(* PLC project Scenario24, Beckhoff Automation GmbH TwinCAT PLC Control 3.5.8.40 *)
(* stored: creationDateTime 2018-05-29T16:20:14.9693905, modificationDateTime 2018-05-29T16:20:14.9929599 *)

TYPE RFID_ByteArray :
STRUCT
	RFID_Data : ARRAY[0..127] OF BYTE;
END_STRUCT
END_TYPE

PROGRAM MAIN
VAR		
	xPPU : xPPU;

//Stack
	//Waiting for Signals
	Check_Stack_WPPickedUp :BOOL;	
	//Giving Signals
	Stack_WPProvided : BOOL;
	Stack_WPType_Black : BOOL;
	Stack_WPType_White : BOOL;
	Stack_WPType_Metallic : BOOL;
	Stack_WPWeight_Light : BOOL;
	Stack_WPWeight_Medium : BOOL;
	Stack_WPWeight_Heavy : BOOL;
//Crane
	//Waiting for Signals
	Check_Stack_WPProvided : BOOL;
	Check_Stack_WPType_Black : BOOL;
	Check_Stack_WPType_White : BOOL;
	Check_Stack_WPType_Metallic : BOOL;
	Check_LargeSortingConveyor_IsSorting : BOOL;
	Check_LargeSortingConveyor_AutomaticExecuteCompleted : BOOL;	
	Check_Stamp_IsStamping : BOOL;
	Check_Stamp_WPAvailable : BOOL;
	Check_Stamp_AutomaticExecuteCompleted : BOOL;
	Check_RefillConveyor_IsSending : BOOL;
	//Giving Signals
	Crane_WPType_Black : BOOL;
	Crane_WPType_White : BOOL;
	Crane_WPType_Metallic : BOOL;
	Crane_WPWeight_Light : BOOL;
	Crane_WPWeight_Medium : BOOL;
	Crane_WPWeight_Heavy : BOOL;
	Crane_Conveyor_AllowedToOperate : BOOL;
	Crane_Stamp_AllowedToOperate : BOOL;
	Crane_WPPickedUp : BOOL;
//Stamp	
	//Waiting for Signals
	Check_Stamp_AllowedToOperate : BOOL;
	Check_Stamp_WPWeight_Light : BOOL;
	Check_Stamp_WPWeight_Medium : BOOL;
    Check_Stamp_WPWeight_Heavy : BOOL;
	//Giving Signals
	Stamp_WPType_Black : BOOL;
	Stamp_WPType_White : BOOL;
	Stamp_WPType_Metallic : BOOL;
	Stamp_WPWeight_Light : BOOL;
	Stamp_WPWeight_Medium : BOOL;
	Stamp_WPWeight_Heavy : BOOL;
	Stamp_IsStamping : BOOL;
	Stamp_WPAvailable : BOOL;
	Stamp_AutomaticExecuteCompleted	: BOOL;
//LargeSortingConveyor
	//Waiting for Signals
	Check_LargeSortingConveyor_AllowedToOperate : BOOL;
	Check_LargeSortingConveyor_FollowConveyorInitCompleted : BOOL;	
	Check_LargeSortingConveyor_FollowConveyorAutoamticExecuteCompleted : BOOL;	
	//Giving Signals	
	LargeSortingConveyor_InitCompleted : BOOL;
	LargeSortingConveyor_NumberOfWPsAtConveyor : USINT;
	LargeSortingConveyor_FollowConveyor_AllowedToInit : BOOL;
	LargeSortingConveyor_FollowConveyor_AllowedToOperate: BOOL;
	LargeSortingConveyor_IsSorting : BOOL;
	LargeSortingConveyor_AutomaticExecuteCompleted : BOOL;	
//PicALphaConveyor
	//Waiting for Signals
	Check_PicAlphaConveyor_AllowedToInit : BOOL;
	Check_PicAlphaConveyor_AllowedToReceive : BOOL;
	Check_PicAlphaConveyor_AllowedToSend : BOOL;
	Check_PicAlphaConveyor_FollowConveyor_InitCompleted : BOOL;
	Check_PicAlphaConveyor_PicAlpha_AutomaticExecuteCompleted : BOOL;
	Check_PicAlphaConveyor_FollowConveyor_AutomaticExecuteCompleted : BOOL;
	//Giving Signals
	PicAlphaConveyor_InitCompleted : BOOL;
	PicAlphaConveyor_FollowConveyor_AllowedToInit : BOOL;
	PicAlphaConveyor_PicAlpha_AllowedToOperate : BOOL;
	PicAlphaConveyor_FollowConveyor_AllowedToOperate: BOOL;
	PicAlphaConveyor_AutomaticExecuteReceivingCompleted : BOOL;
	PicAlphaConveyor_AutomaticExecuteSendingCompleted : BOOL;
//SmallSortingConveyor
	//Waiting for Signals
	Check_SmallSortingConveyor_AllowedToInit : BOOL;
	Check_SmallSortingConveyor_AllowedToOperate : BOOL;	
	Check_SmallSortingConveyor_FollowConveyor_InitCompleted : BOOL;
	Check_SmallSortingConveyor_FollowConveyor_AutomaticExecuteCompleted : BOOL;
	//Giving Signals
	SmallSortingConveyor_InitCompleted : BOOL;
	SmallSortingConveyor_FollowConveyor_AllowedToInit : BOOL;
	SmallSortingConveyor_FollowConveyor_AllowedToOperate: BOOL;
	SmallSortingConveyor_AutomaticExecuteCompleted : BOOL;
	SmallSortingConveyor_IsSorting : BOOL;	
//RefillConveyor
	//Waiting for Signals
	Check_RefillConveyor_AllowedToInit : BOOL;
	Check_RefillConveyor_AllowedToReceive : BOOL;
	Check_RefillConveyor_AllowedToSend : BOOL;
	Check_RefillConveyor_FollowConveyor_InitCompleted : BOOL;
	Check_RefillConveyor_FollowConveyor_AutomaticExecuteCompleted : BOOL;
	//Giving Signals
	RefillConveyor_InitCompleted : BOOL;
	RefillConveyor_FollowConveyor_AllowedToInit : BOOL;
	RefillConveyor_FollowConveyor_AllowedToOperate: BOOL;
	RefillConveyor_AutomaticExecuteReceivingCompleted : BOOL;
	RefillConveyor_IsSending : BOOL;
	RefillConveyor_AutomaticExecuteSendingCompleted : BOOL;	
//PicAlpha
	//Waiting for Signals
	Check_PicAlpha_AllowedToOperate : BOOL;
	Check_PicAlpha_Conveyor_AutomaticExecuteCompleted : BOOL;
	//Giving Signals
	PicAlpha_InitCompleted : BOOL;
	PicAlpha_Conveyor_AllowedToOperate : BOOL;
	PicAlpha_AutomaticExecuteCompleted : BOOL;
//PPU
	PPU_EngineStop : BOOL;
END_VAR

                  xPPU();
xPPU.Stack();
xPPU.Crane();
xPPU.Stamp();
xPPU.LargeSortingConveyor();
xPPU.PicAlphaConveyor();
xPPU.SmallSortingConveyor();
xPPU.RefillConveyor();
xPPU.PicAlpha();
xPPU.SafetyDoor();
xPPU.LightGrid();


//Stack
	//Waiting for Signals
	Check_Stack_WPPickedUp := xPPU.Crane.Table.AtStack.DI_SwitchTrue AND xPPU.Crane.WPPickedUp;	
	//Giving Signals
	Stack_WPProvided := xPPU.Stack.WPProvided;
	Stack_WPType_Black := xPPU.Stack.WPType_Black;
	Stack_WPType_White := xPPU.Stack.WPType_White;
	Stack_WPType_Metallic := xPPU.Stack.WPType_Metallic;
	Stack_WPWeight_Light := xPPU.Stack.WPWeight_Light;
	Stack_WPWeight_Medium := xPPU.Stack.WPWeight_Medium;
	Stack_WPWeight_Heavy := xPPU.Stack.WPWeight_Heavy;	
//Crane
	//Waiting for Signals
	Check_Stack_WPProvided := Stack_WPProvided;
	Check_Stack_WPType_Black := Stack_WPType_Black;
	Check_Stack_WPType_White := Stack_WPType_White;
	Check_Stack_WPType_Metallic := Stack_WPType_Metallic;
	Check_LargeSortingConveyor_IsSorting := LargeSortingConveyor_IsSorting;
	Check_LargeSortingConveyor_AutomaticExecuteCompleted := LargeSortingConveyor_AutomaticExecuteCompleted;	
	Check_Stamp_IsStamping := Stamp_IsStamping;
	Check_Stamp_WPAvailable := Stamp_WPAvailable;
	Check_Stamp_AutomaticExecuteCompleted := Stamp_AutomaticExecuteCompleted;
	Check_RefillConveyor_IsSending := RefillConveyor_IsSending;
	//Giving Signals
	Crane_WPType_Black := xPPU.Crane.WPType_Black;
	Crane_WPType_White := xPPU.Crane.WPType_White;
	Crane_WPType_Metallic := xPPU.Crane.WPType_Metallic;
	Crane_WPWeight_Light := xPPU.Crane.WPWeight_Light;
	Crane_WPWeight_Medium := xPPU.Crane.WPWeight_Medium;
	Crane_WPWeight_Heavy := xPPU.Crane.WPWeight_Heavy;
	Crane_Conveyor_AllowedToOperate := xPPU.Crane.Conveyor_AllowedToOperate;
	Crane_Stamp_AllowedToOperate := xPPU.Crane.Stamp_AllowedToOperate;
	Crane_WPPickedUp := xPPU.Crane.Gripper.VacuumSwitch.DI_TakenIn;
//Stamp	
	//Waiting for Signals
	Check_Stamp_AllowedToOperate := Crane_Stamp_AllowedToOperate;
	Check_Stamp_WPWeight_Light := Crane_WPWeight_Light;
	Check_Stamp_WPWeight_Medium := Crane_WPWeight_Medium;
    Check_Stamp_WPWeight_Heavy := Crane_WPWeight_Heavy;
	//Giving Signals
	Stamp_WPType_Black := xPPU.Stamp.WPType_Black;
	Stamp_WPType_White := xPPU.Stamp.WPType_White;
	Stamp_WPType_Metallic := xPPU.Stamp.WPType_Metallic;
	Stamp_WPWeight_Light := xPPU.Stamp.WPWeight_Light;
	Stamp_WPWeight_Medium := xPPU.Stamp.WPWeight_Medium;
	Stamp_WPWeight_Heavy := xPPU.Stamp.WPWeight_Heavy;
	Stamp_IsStamping := xPPU.Stamp.IsStamping;
	Stamp_WPAvailable := xPPU.Stamp.WPAvailable.DI_SwitchTrue;
	Stamp_AutomaticExecuteCompleted	:= xPPU.Stamp.AutomaticExecuteCompleted;
//LargeSortingConveyor
	//Waiting for Signals
	Check_LargeSortingConveyor_AllowedToOperate := Crane_Conveyor_AllowedToOperate OR RefillConveyor_FollowConveyor_AllowedToOperate;
	Check_LargeSortingConveyor_FollowConveyorInitCompleted := PicALphaConveyor_InitCompleted;	
	Check_LargeSortingConveyor_FollowConveyorAutoamticExecuteCompleted := PicALphaConveyor_AutomaticExecuteReceivingCompleted;	
	//Giving Signals
	LargeSortingConveyor_NumberOfWPsAtConveyor := xPPU.LargeSortingConveyor.NumberOfWPsAtConveyor;
	LargeSortingConveyor_FollowConveyor_AllowedToInit := xPPU.LargeSortingConveyor.FollowConveyor_AllowedToInit;
	LargeSortingConveyor_FollowConveyor_AllowedToOperate:= xPPU.LargeSortingConveyor.FollowConveyor_AllowedToOperate;
	LargeSortingConveyor_IsSorting := xPPU.LargeSortingConveyor.IsSorting;
	LargeSortingConveyor_AutomaticExecuteCompleted := xPPU.LargeSortingConveyor.AutomaticExecuteCompleted;	
//PicALphaConveyor
	//Waiting for Signals
	Check_PicAlphaConveyor_AllowedToInit := LargeSortingConveyor_FollowConveyor_AllowedToInit;
	Check_PicAlphaConveyor_AllowedToReceive := LargeSortingConveyor_FollowConveyor_AllowedToOperate;
	Check_PicAlphaConveyor_AllowedToSend := LargeSortingConveyor_NumberOfWPsAtConveyor=3;
	Check_PicAlphaConveyor_FollowConveyor_InitCompleted := SmallSortingConveyor_InitCompleted;
	Check_PicAlphaConveyor_PicAlpha_AutomaticExecuteCompleted := PicAlpha_AutomaticExecuteCompleted;
	Check_PicAlphaConveyor_FollowConveyor_AutomaticExecuteCompleted := SmallSortingConveyor_AutomaticExecuteCompleted;
	//Giving Signals
	PicAlphaConveyor_InitCompleted := xPPU.PicALphaConveyor.InitCompleted;
	PicAlphaConveyor_FollowConveyor_AllowedToInit := xPPU.PicALphaConveyor.FollowConveyor_AllowedToInit;
	PicAlphaConveyor_PicAlpha_AllowedToOperate := xPPU.PicAlphaConveyor.PicAlpha_AllowedToOperate;
	PicAlphaConveyor_FollowConveyor_AllowedToOperate := xPPU.PicALphaConveyor.FollowConveyor_AllowedToOperate;
	PicAlphaConveyor_AutomaticExecuteReceivingCompleted := xPPU.PicALphaConveyor.AutomaticExecuteReceivingCompleted;
	PicAlphaConveyor_AutomaticExecuteSendingCompleted := xPPU.PicALphaConveyor.AutomaticExecuteSendingCompleted;
//SmallSortingConveyor
	//Waiting for Signals
	Check_SmallSortingConveyor_AllowedToInit := PicALphaConveyor_FollowConveyor_AllowedToInit;
	Check_SmallSortingConveyor_AllowedToOperate := PicALphaConveyor_FollowConveyor_AllowedToOperate;	
	Check_SmallSortingConveyor_FollowConveyor_InitCompleted := RefillConveyor_InitCompleted;
	Check_SmallSortingConveyor_FollowConveyor_AutomaticExecuteCompleted := RefillConveyor_AutomaticExecuteReceivingCompleted;
	//Giving Signals
	SmallSortingConveyor_InitCompleted := xPPU.SmallSortingConveyor.InitCompleted;
	SmallSortingConveyor_FollowConveyor_AllowedToInit := xPPU.SmallSortingConveyor.FollowConveyor_AllowedToInit;
	SmallSortingConveyor_FollowConveyor_AllowedToOperate:= xPPU.SmallSortingConveyor.FollowConveyor_AllowedToOperate;
	SmallSortingConveyor_AutomaticExecuteCompleted := xPPU.SmallSortingConveyor.AutomaticExecuteCompleted;
	SmallSortingConveyor_IsSorting := xPPU.SmallSortingConveyor.IsSorting;	
//RefillConveyor
	//Waiting for Signals
	Check_RefillConveyor_AllowedToInit := SmallSortingConveyor_FollowConveyor_AllowedToInit;
	Check_RefillConveyor_AllowedToReceive := SmallSortingConveyor_FollowConveyor_AllowedToOperate;
	Check_RefillConveyor_AllowedToSend := NOT Crane_WPPickedUp AND NOT LargeSortingConveyor_IsSorting AND NOT Check_LargeSortingConveyor_AllowedToOperate;
	Check_RefillConveyor_FollowConveyor_InitCompleted := LargeSortingConveyor_InitCompleted;
	Check_RefillConveyor_FollowConveyor_AutomaticExecuteCompleted := LargeSortingConveyor_AutomaticExecuteCompleted;
	//Giving Signals
	RefillConveyor_InitCompleted := xPPU.RefillConveyor.InitCompleted;
	RefillConveyor_FollowConveyor_AllowedToInit := xPPU.RefillConveyor.FollowConveyor_AllowedToInit;
	RefillConveyor_FollowConveyor_AllowedToOperate := xPPU.RefillConveyor.FollowConveyor_AllowedToOperate;
	RefillConveyor_AutomaticExecuteReceivingCompleted := xPPU.RefillConveyor.AutomaticExecuteReceivingCompleted;
	RefillConveyor_IsSending := xPPU.RefillConveyor.IsSending;
	RefillConveyor_AutomaticExecuteSendingCompleted := xPPU.RefillConveyor.AutomaticExecuteSendingCompleted;	
//PicAlpha
	//Waiting for Signals
	Check_PicAlpha_AllowedToOperate := PicAlphaConveyor_PicAlpha_AllowedToOperate;
	Check_PicAlpha_Conveyor_AutomaticExecuteCompleted := PicAlphaConveyor_AutomaticExecuteSendingCompleted;
	//Giving Signals
	PicAlpha_InitCompleted := xPPU.PicAlpha.InitCompleted;
	PicAlpha_Conveyor_AllowedToOperate := xPPU.PicAlpha.Conveyor_AllowedToOperate;
//PPU
	PPU_EngineStop := xPPU.ManuelMode;	
	
	
	
	

	PicAlpha_AutomaticExecuteCompleted := xPPU.PicAlpha.AutomaticExecuteCompleted;		
                
END_PROGRAM

FUNCTION_BLOCK BistableCylinder
VAR_INPUT	
END_VAR
VAR_OUTPUT
	//Software
	Extended : BOOL;
	Retracted : BOOL;
END_VAR
VAR	
	//Hardware
	DI_Extended AT %I* : BOOL;
	DI_Retracted AT %I* : BOOL;	
	DO_Extend AT %Q* : BOOL;
	DO_Retract AT %Q* : BOOL;
	//NOT USED BUT USABLE 
	DI_BoundaryPressure AT %I* : BOOL;
	DI_VacuumBoundaryPressure AT %I* : BOOL;
	DI_VacuumBoundaryFlowPressure AT %I* : BOOL;
	AI_PressureSensor AT %I* : INT;
	AI_FlowPressure AT %I* : INT;	
	AI_PositionTransmitter AT %I* : INT;
END_VAR

                  
                

ACTION ACT_Extend:
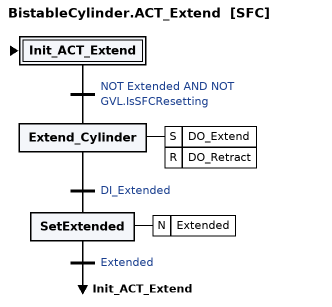
INITIAL_STEP Init_ACT_Extend:
END_STEP
TRANSITION FROM Init_ACT_Extend TO Extend_Cylinder
  := NOT Extended AND NOT GVL.IsSFCResetting;
END_TRANSITION
STEP Extend_Cylinder:
  DO_Extend(S);
  DO_Retract(R);
END_STEP
TRANSITION FROM Extend_Cylinder TO SetExtended
  := DI_Extended;
END_TRANSITION
STEP SetExtended:
  Extended(N);
END_STEP
TRANSITION FROM SetExtended TO Init_ACT_Extend
  := Extended;
END_TRANSITION
END_ACTION

ACTION ACT_Retract:
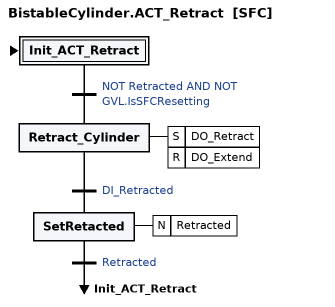
INITIAL_STEP Init_ACT_Retract:
END_STEP
TRANSITION FROM Init_ACT_Retract TO Retract_Cylinder
  := NOT Retracted AND NOT GVL.IsSFCResetting;
END_TRANSITION
STEP Retract_Cylinder:
  DO_Retract(S);
  DO_Extend(R);
END_STEP
TRANSITION FROM Retract_Cylinder TO SetRetacted
  := DI_Retracted;
END_TRANSITION
STEP SetRetacted:
  Retracted(N);
END_STEP
TRANSITION FROM SetRetacted TO Init_ACT_Retract
  := Retracted;
END_TRANSITION
END_ACTION
END_FUNCTION_BLOCK

FUNCTION_BLOCK InductiveSensor
VAR_INPUT
END_VAR
VAR_OUTPUT
END_VAR
VAR
	//Hardware
	DI_WPMetallic AT %I* : BOOL;
END_VAR

                  
                
END_FUNCTION_BLOCK

FUNCTION_BLOCK InductiveSwitch
VAR_INPUT
END_VAR
VAR_OUTPUT
END_VAR
VAR
	//Hardware
	DI_InductiveSwitchTrue AT %I* : BOOL;
END_VAR

                  
                
END_FUNCTION_BLOCK

FUNCTION_BLOCK MicroSwitch
VAR_INPUT
END_VAR
VAR_OUTPUT
END_VAR
VAR
	//Hardware
	DI_SwitchTrue AT %I* : BOOL;
END_VAR

                  
                
END_FUNCTION_BLOCK

FUNCTION_BLOCK MonostableCylinder
VAR_INPUT	
END_VAR	
VAR_OUTPUT	
	//Software
	Extended : BOOL;
	Retracted : BOOL;
END_VAR
VAR	
	//Hardware
	DI_Extended AT %I* : BOOL;
	DI_Retracted AT %I* : BOOL;	
	DO_Extend AT %Q* : BOOL;
	//NOT USED BUT USABLE	
	DI_BoundaryPressure AT %I* : BOOL;
	DI_BoundaryFlowPressure AT %I* : BOOL;
	AI_PressureSensor AT %I* : INT;
	AI_FlowPressure AT %I* : INT;
	AI_PositionTransmitter AT %I* : INT;
END_VAR

                  
                

ACTION ACT_Extend:
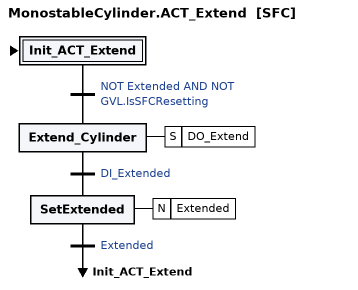
INITIAL_STEP Init_ACT_Extend:
END_STEP
TRANSITION FROM Init_ACT_Extend TO Extend_Cylinder
  := NOT Extended AND NOT GVL.IsSFCResetting;
END_TRANSITION
STEP Extend_Cylinder:
  DO_Extend(S);
END_STEP
TRANSITION FROM Extend_Cylinder TO SetExtended
  := DI_Extended;
END_TRANSITION
STEP SetExtended:
  Extended(N);
END_STEP
TRANSITION FROM SetExtended TO Init_ACT_Extend
  := Extended;
END_TRANSITION
END_ACTION

ACTION ACT_Retract:
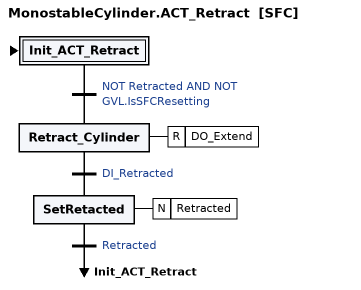
INITIAL_STEP Init_ACT_Retract:
END_STEP
TRANSITION FROM Init_ACT_Retract TO Retract_Cylinder
  := NOT Retracted AND NOT GVL.IsSFCResetting;
END_TRANSITION
STEP Retract_Cylinder:
  DO_Extend(R);
END_STEP
TRANSITION FROM Retract_Cylinder TO SetRetacted
  := DI_Retracted;
END_TRANSITION
STEP SetRetacted:
  Retracted(N);
END_STEP
TRANSITION FROM SetRetacted TO Init_ACT_Retract
  := Retracted;
END_TRANSITION
END_ACTION
END_FUNCTION_BLOCK

FUNCTION_BLOCK Motor
VAR_INPUT
	//Software
	Stopped : BOOL;
	TurningClockwise : BOOL;
	TurningCounterclockwise : BOOL;
END_VAR
VAR_OUTPUT			
	AI_Position AT %I*: UINT;
	AI_Speed AT %I*: UDINT;
END_VAR
VAR	
	//Hardware
	DO_TurnClockwise AT %Q* : BOOL;
	DO_TurnCounterclockwise AT %Q* : BOOL;	
END_VAR

                  
                

ACTION ACT_Stop:
                      DO_TurnClockwise := FALSE;
DO_TurnCounterclockwise := FALSE;

Stopped := TRUE;
TurningClockwise := FALSE;
TurningCounterclockwise := FALSE;
                    
END_ACTION

ACTION ACT_TurnClockwise:
                      DO_TurnClockwise := TRUE;
DO_TurnCounterclockwise := FALSE;

Stopped := FALSE;
TurningClockwise := TRUE;
TurningCounterclockwise := FALSE;
                    
END_ACTION

ACTION ACT_TurnCounterclockwise:
                      DO_TurnClockwise := FALSE;
DO_TurnCounterclockwise := TRUE;

Stopped := FALSE;
TurningClockwise := FALSE;
TurningCounterclockwise := TRUE;
                    
END_ACTION
END_FUNCTION_BLOCK

FUNCTION_BLOCK OperationPanel
VAR_INPUT
END_VAR
VAR_OUTPUT
	//Software
	EmergencyStop : BOOL;
	StartButton : BOOL;
	ManuelMode : BOOL;
	AutomaticMode : BOOL;
END_VAR
VAR
	//Hardware
	DI_StartButton AT %I* : BOOL;
	DI_AutomaticButton AT %I* : BOOL;	
	DI_EmergencyStop AT %I* : BOOL;	
	DO_LampGreen AT %Q* : BOOL;
	DO_LampWhite AT %Q* : BOOL;
END_VAR

                  EmergencyStop := NOT DI_EmergencyStop;
StartButton := DI_StartButton;
ManuelMode := NOT DI_AutomaticButton;
AutomaticMode := DI_AutomaticButton;
                

ACTION ACT_TurnLampGreen_Off:
                      DO_LampGreen := FALSE;
                    
END_ACTION

ACTION ACT_TurnLampGreen_On:
                      DO_LampGreen := TRUE;
                    
END_ACTION

ACTION ACT_TurnLampWhite_Off:
                      DO_LampWhite:=FALSE;
                    
END_ACTION

ACTION ACT_TurnLampWhite_On:
                      DO_LampWhite:=TRUE;
                    
END_ACTION
END_FUNCTION_BLOCK

FUNCTION_BLOCK OperationPanelExtended
VAR_INPUT
END_VAR
VAR_OUTPUT
	//Software
	EmergencyStop : BOOL;
	StartButton : BOOL;
	ManuelMode : BOOL;
	AutomaticMode : BOOL;
	Reset : BOOL;
END_VAR
VAR
	//Hardware
	DI_EmergencyStop AT %I* : BOOL;
	DI_StartButton AT %I* : BOOL;
	DI_AutomaticButton AT %I* : BOOL;	
	DI_StopButton AT %I* : BOOL;	
	DI_ResetButton AT %I* : BOOL;
	DO_LampGreen AT %Q* : BOOL;
	DO_LampReset AT %Q* : BOOL;
	DO_Q1 AT %Q* : BOOL;
	DO_Q2 AT %Q* : BOOL;
END_VAR

                  EmergencyStop := NOT DI_StopButton;
StartButton := DI_StartButton;
ManuelMode := NOT DI_AutomaticButton;
AutomaticMode := DI_AutomaticButton;
Reset := DI_ResetButton;
                

ACTION ACT_TurnLampGreen_Off:
                      DO_LampGreen := FALSE;
                    
END_ACTION

ACTION ACT_TurnLampGreen_On:
                      DO_LampGreen := TRUE;
                    
END_ACTION

ACTION ACT_TurnLampReset_Off:
                      DO_LampReset:=FALSE;
                    
END_ACTION

ACTION ACT_TurnLampReset_On:
                      DO_LampReset:=TRUE;
                    
END_ACTION
END_FUNCTION_BLOCK

FUNCTION_BLOCK OpticalSensor
VAR_INPUT
END_VAR
VAR_OUTPUT
END_VAR
VAR
	//Hardware
	DI_WPLight AT %I* : BOOL;
END_VAR

                  
                
END_FUNCTION_BLOCK

FUNCTION_BLOCK PositionTransmitter
VAR_INPUT
END_VAR
VAR_OUTPUT
	//Hardware
	DI_PositionReached AT %I* : BOOL; 
END_VAR
VAR
END_VAR

                  
                
END_FUNCTION_BLOCK

FUNCTION_BLOCK Potentiometer
VAR_INPUT
END_VAR
VAR_OUTPUT
	//Software	
	AtStack : BOOL;
	AtStackRFID : BOOL;
	AtConveyor : BOOL;
	AtConveyorRFID : BOOL;
	AtStamp : BOOL;
	AtStampRFID : BOOL;
END_VAR
VAR
	//Hardware
	AI_Position AT%I* : INT;
	//Software
	delta : INT := 150;
	iPosStack : INT := 24310;
	iPosStackRFID : INT := 23290;
	iPosConveyor : INT := 15930;
	iPosConveyorRFID : INT := 14890;
	iPosStamp : INT := 7845;
	iPosStampRFID : INT := 6810;
END_VAR

                  IF((iPosStack-delta) < AI_Position AND AI_Position < (iPosStack+delta)) THEN //AT STACK
	AtStack := TRUE;
	AtStackRFID := FALSE;
	AtConveyor := FALSE;
	AtConveyorRFID := FALSE;
	AtStamp := FALSE;
	AtStampRFID := FALSE;
ELSIF((iPosStackRFID-delta) < AI_Position AND AI_Position < (iPosStackRFID+delta)) THEN //AT STACK RFID	
	AtStack := FALSE;
	AtStackRFID := TRUE;
	AtConveyor := FALSE;
	AtConveyorRFID := FALSE;
	AtStamp := FALSE;
	AtStampRFID := FALSE;
ELSIF((iPosConveyor-delta) < AI_Position AND AI_Position < (iPosConveyor+delta)) THEN //AT CONVEYOR
	AtStack := FALSE;
	AtStackRFID := FALSE;
	AtConveyor := TRUE;
	AtConveyorRFID := FALSE;
	AtStamp := FALSE;
	AtStampRFID := FALSE;
ELSIF((iPosConveyorRFID-delta) < AI_Position AND AI_Position < (iPosConveyorRFID+delta)) THEN //AT CONVEYOR RFID
	AtStack := FALSE;
	AtStackRFID := FALSE;
	AtConveyor := FALSE;
	AtConveyorRFID := TRUE;
	AtStamp := FALSE;
	AtStampRFID := FALSE;
ELSIF((iPosStamp-delta) < AI_Position AND AI_Position < (iPosStamp+delta)) THEN //AT STAMP
	AtStack := FALSE;
	AtStackRFID := FALSE;
	AtConveyor := FALSE;
	AtConveyorRFID := FALSE;
	AtStamp := TRUE;
	AtStampRFID := FALSE;
ELSIF((iPosStampRFID-delta) < AI_Position AND AI_Position < (iPosStampRFID+delta)) THEN //AT STAMP RFIG
	AtStack := FALSE;
	AtStackRFID := FALSE;
	AtConveyor := FALSE;
	AtConveyorRFID := FALSE;
	AtStamp := FALSE;
	AtStampRFID := TRUE;
ELSE
	AtStack := FALSE;
	AtStackRFID := FALSE;
	AtConveyor := FALSE;
	AtConveyorRFID := FALSE;
	AtStamp := FALSE;
	AtStampRFID := FALSE;	
END_IF
                
END_FUNCTION_BLOCK

FUNCTION_BLOCK PresenceSensor
VAR_INPUT
END_VAR
VAR_OUTPUT
END_VAR
VAR
	DI_WPDetected AT %I* : BOOL;
END_VAR

                  
                
END_FUNCTION_BLOCK

FUNCTION_BLOCK PressureSensor
VAR_INPUT
END_VAR
VAR_OUTPUT
END_VAR
VAR
	//Hardware
	AI_CurrentPressure AT %I* : INT;
END_VAR

                  
                
END_FUNCTION_BLOCK

FUNCTION_BLOCK ProportionalValve
VAR_INPUT
	//Hardware
	AO_SetPressure AT %Q* : INT;
END_VAR
VAR_OUTPUT
END_VAR
VAR	
END_VAR

                  
                
END_FUNCTION_BLOCK

FUNCTION_BLOCK Ramp
VAR_INPUT
	//Hardware
	RampFull : PresenceSensor;
END_VAR
VAR_OUTPUT
END_VAR
VAR
END_VAR

                  
                
END_FUNCTION_BLOCK

FUNCTION_BLOCK RFID
VAR_INPUT
	Data_to_Write : RFID_ByteArray;
	bRead : BOOL;
	bWrite : BOOL;
	bAntOFF : BOOL;
	bAntON : BOOL;
END_VAR
VAR_OUTPUT
	RFID_Status : BYTE;
	Error_Number : BYTE;
	Error_Code : WSTRING;
	Done_Writing : BOOL;
	Done_Reading : BOOL;
	Done_Resetting : BOOL;
	Data_Last_RFID : RFID_ByteArray; 
END_VAR
VAR	
	//Hardware
	//PAE 
	AI_Status AT%I* : BYTE; //IO_Link Port2_in UID Byte 0
	AI_error_RFID AT%I* : BYTE; //IO_Link Port2_in UID Byte 1
	AI_Adr_H AT%I* : BYTE; //IO_Link Port2_in UID Byte 2
	AI_Adr_L AT%I* : BYTE; //IO_Link Port2_in UID Byte 3
	AI_Data_MSB AT%I* : BYTE; //IO_Link Port2_in UID Byte 4
	AI_Data_5 AT%I* : BYTE; //IO_Link Port2_in UID Byte 5
	AI_Data_6 AT%I* : BYTE; //IO_Link Port2_in UID Byte 6
	AI_Data_LSB AT%I* : BYTE; //IO_Link Port2_in UID Byte 7
	//PAA
	AO_CMD AT%Q* : BYTE; //IO_Link Port2_out Antenne
	AO_Adr_H AT%Q* : BYTE; //IO_Link Port2_out Reserved_1
	AO_Adr_L AT%Q* : BYTE; //IO_Link Port2_out Reserved_2
	AO_Data_MSB AT%Q* : BYTE; //IO_Link Port2_out Reserved_3
	AO_Data_5 AT%Q* : BYTE; //IO_Link Port2_out Reserved_4
	AO_Data_6 AT%Q* : BYTE; //IO_Link Port2_out Reserved_5
	AO_Data_LSB AT%Q* : BYTE; //IO_Link Port2_out Reserved_6
	
	//Process Image Input
	StausByte_CommandCode_0 : BOOL; //WRITE
	StausByte_CommandCode_1 : BOOL; //READ
	StausByte_CommandCode_2: BOOL;
	StausByte_CommandCode_3 : BOOL;
	StausByte_ANT_OFF_Conf : BOOL;
	StatusByte_RFID_Present : BOOL;
	StatusByte_ErrorOccured : BOOL;
	StatusByte_Command_executed : BOOL;
	
	//Software
	//Provces Image Output
	CMD_Write : BYTE := 2#0000_0001;	
	CMD_Read : BYTE := 2#0000_0010;	
	CMD_Antenna_Off : BYTE := 2#0001_0000;
	CMD_Antenna_On : BYTE := 2#0000_0000;
	
 		
	Step : INT := 10;
	Counter : UINT;
	TagData : RFID_ByteArray; 
	
	DataToWriteCounter : INT;
END_VAR

                  ACT_ConvertStatusByteToBits();
ACT_ErrorCodeTranslation();
                

ACTION ACT_AntennaOFF:
                      AO_CMD := CMD_Antenna_Off;
                    
END_ACTION

ACTION ACT_AntennaON:
                      AO_CMD := CMD_Antenna_On;
                    
END_ACTION

ACTION ACT_ConvertStatusByteToBits:
                      //Bit 0
IF((AI_Status AND 1)=1) THEN
	StausByte_CommandCode_0 := TRUE;
ELSE
	StausByte_CommandCode_0 := FALSE;
END_IF
//Bit 1
IF((AI_Status AND 2)=2) THEN
	StausByte_CommandCode_1 := TRUE;
ELSE
	StausByte_CommandCode_1 := FALSE;
END_IF
//Bit 2
IF((AI_Status AND 4)=4) THEN
	StausByte_CommandCode_2 := TRUE;
ELSE
	StausByte_CommandCode_2 := FALSE;
END_IF
//Bit 3
IF((AI_Status AND 8)=8) THEN
	StausByte_CommandCode_3 := TRUE;
ELSE
	StausByte_CommandCode_3 := FALSE;
END_IF
//Bit 4
IF((AI_Status AND 16)=16) THEN
	StausByte_ANT_OFF_Conf := TRUE;
ELSE
	StausByte_ANT_OFF_Conf := FALSE;
END_IF
//Bit 5
IF((AI_Status AND 32)=32) THEN
	StatusByte_RFID_Present := TRUE;
ELSE
	StatusByte_RFID_Present := FALSE;
END_IF
//Bit 6
IF((AI_Status AND 64)=64) THEN
	StatusByte_ErrorOccured := TRUE;
ELSE
	StatusByte_ErrorOccured := FALSE;
END_IF
//Bit 7
IF((AI_Status AND 128)=128) THEN
	StatusByte_Command_executed := TRUE;
ELSE
	StatusByte_Command_executed := FALSE;
END_IF
                    
END_ACTION

ACTION ACT_CreateDataToWirte:
                      //Write 0 at every Position (Deleting old Data)
IF(DataToWriteCounter<=127)THEN
	Data_to_Write.RFID_Data[DataToWriteCounter]:= INT_TO_BYTE(0);
	DataToWriteCounter := DataToWriteCounter +1;
END_IF
//Write on specified position specified data (here Pos:= 10, Value:=1)
Data_to_Write.RFID_Data[2]:= INT_TO_BYTE(1);
                    
END_ACTION

ACTION ACT_ErrorCodeTranslation:
                      Error_Number:=AI_error_RFID;

//Fehlercodeauswertung
IF(Error_Number=0)THEN
	Error_Code := "no Error";
ELSIF(Error_Number=1)THEN	
	Error_Code := "Presence Error";	
ELSIF(Error_Number=5)THEN	
	Error_Code := "Parameterization Error";	
ELSIF(Error_Number=6)THEN	
	Error_Code := "Air interface disturbed";
ELSIF(Error_Number=12)THEN	
	Error_Code := "Memory Error";
ELSIF(Error_Number=13)THEN	
	Error_Code := "Error with the indicated storage adress";	
ELSIF(Error_Number=19)THEN	
	Error_Code := "Buffer Overflow";
ELSIF(Error_Number=20)THEN	
	Error_Code := "Serious System Error";
ELSIF(Error_Number=21)THEN	
	Error_Code := "Parameterization Error in the RESET-Command";
ELSIF(Error_Number=24)THEN	
	Error_Code := "Only RESET-Command allowed";
ELSIF(Error_Number=25)THEN	
	Error_Code := "Previous command is still active";
ELSIF(Error_Number=28)THEN	
	Error_Code := "Antenna is allready ON/OFF";
ELSIF(Error_Number=30)THEN	
	Error_Code := "Wronge number of signs in the telegram";
END_IF
                    
END_ACTION

ACTION ACT_Read_Write_Test:
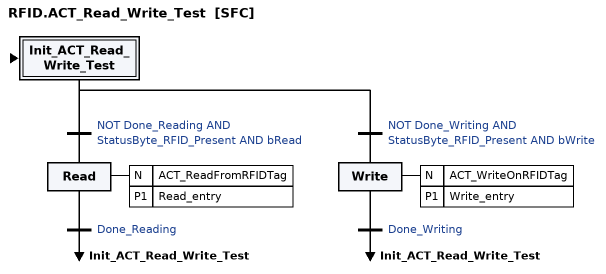
INITIAL_STEP Init_ACT_Read_Write_Test:
END_STEP
TRANSITION FROM Init_ACT_Read_Write_Test TO Read
  := NOT Done_Reading AND StatusByte_RFID_Present AND bRead;
END_TRANSITION
TRANSITION FROM Init_ACT_Read_Write_Test TO Write
  := NOT Done_Writing AND StatusByte_RFID_Present AND bWrite;
END_TRANSITION
STEP Read:
  ACT_ReadFromRFIDTag(N);
  Read_entry(P1);
END_STEP
TRANSITION FROM Read TO Init_ACT_Read_Write_Test
  := Done_Reading;
END_TRANSITION
STEP Write:
  ACT_WriteOnRFIDTag(N);
  Write_entry(P1);
END_STEP
TRANSITION FROM Write TO Init_ACT_Read_Write_Test
  := Done_Writing;
END_TRANSITION
END_ACTION

ACTION ACT_ReadFromRFIDTag:
                      CASE Step OF 
	100:// copy complete Data to internal Array // Set Loop-Counter to 0
		Counter := 0;
		Step := 110;	        
	        
	110:// Read 4 Byte  // Wait until read done
		AO_Adr_L := INT_TO_BYTE(Counter); 
		AO_CMD := CMD_Read;
 
		IF(StatusByte_Command_executed AND StausByte_CommandCode_1)  THEN 		
			Step := 120;			
		END_IF;	        

	120: //copy data and reset command   
		Data_Last_RFID.RFID_Data[Counter]   := AI_Data_LSB;
		Data_Last_RFID.RFID_Data[Counter+1] := AI_Data_6;
		Data_Last_RFID.RFID_Data[Counter+2] := AI_Data_5;
		Data_Last_RFID.RFID_Data[Counter+3] := AI_Data_MSB;
		AO_CMD := CMD_Antenna_On;
		Step := 130;

	130: // Wait until Last command1 is false
		IF (NOT StausByte_CommandCode_1) THEN 
			Step := 140;
		END_IF;	        
	        
    140: // increment counter // compare, if last dword copied
        Counter := Counter + 4;
	    IF(Counter >= 100) THEN
			Step := 150;
        ELSE
            Step := 110;
		END_IF;
	        
    150: // copy complete array back to data // set done = true
        Done_Reading := TRUE;
        Step := 10;
END_CASE





                    
END_ACTION

ACTION ACT_ResetRFID:
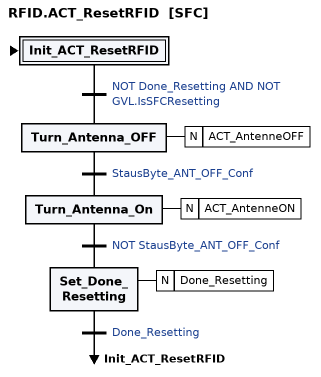
INITIAL_STEP Init_ACT_ResetRFID:
END_STEP
TRANSITION FROM Init_ACT_ResetRFID TO Turn_Antenna_OFF
  := NOT Done_Resetting AND NOT GVL.IsSFCResetting;
END_TRANSITION
STEP Turn_Antenna_OFF:
  ACT_AntenneOFF(N);
END_STEP
TRANSITION FROM Turn_Antenna_OFF TO Turn_Antenna_On
  := StausByte_ANT_OFF_Conf;
END_TRANSITION
STEP Turn_Antenna_On:
  ACT_AntenneON(N);
END_STEP
TRANSITION FROM Turn_Antenna_On TO Set_Done_Resetting
  := NOT StausByte_ANT_OFF_Conf;
END_TRANSITION
STEP Set_Done_Resetting:
  Done_Resetting(N);
END_STEP
TRANSITION FROM Set_Done_Resetting TO Init_ACT_ResetRFID
  := Done_Resetting;
END_TRANSITION
END_ACTION

ACTION ACT_WriteOnRFIDTag:
                      CASE Step OF 
	200:// copy complete Data to internal Array // Set Loop-Counter to 0
		Counter := 0;
		Step := 210;	        
	        
	210:// Write 4 Byte  // Wait until write done
		AO_Adr_L := INT_TO_BYTE(Counter); 
		AO_Data_LSB := Data_to_Write.RFID_Data[Counter];
		AO_Data_6   := Data_to_Write.RFID_Data[Counter+1];
		AO_Data_5   := Data_to_Write.RFID_Data[Counter+2];
		AO_Data_MSB := Data_to_Write.RFID_Data[Counter+3];
		AO_CMD := CMD_Write;
 
		IF(StatusByte_Command_executed AND StausByte_CommandCode_0)  THEN 		
			Step := 220;			
		END_IF;	        

	220: // reset command    
		AO_CMD := CMD_Antenna_On;
		Step := 230;

	230: // Wait until Last command0 is false
		IF (NOT StausByte_CommandCode_0) THEN 
			Step := 240;
		END_IF;	        
	        
    240: // increment counter // compare, if last dword copied
        Counter := Counter + 4;
	    IF(Counter >= 100) THEN
			Step := 250;
        ELSE
            Step := 210;
		END_IF;
	        
    250: // copy complete array back to data // set done = true
        Done_Writing := TRUE;
        Step := 10;
END_CASE
                    
END_ACTION

ACTION Read_entry:
                      Step := 100;
                    
END_ACTION

ACTION Write_entry:
                      Step := 200;
                    
END_ACTION
END_FUNCTION_BLOCK

FUNCTION_BLOCK Switch
VAR_INPUT
END_VAR
VAR_OUTPUT
	//Software
	Extended : BOOL;
	Retracted : BOOL;
END_VAR
VAR
	//Hardware
	DI_Extended AT %I* : BOOL;
	DI_Retracted AT %I* : BOOL;	
	DO_Extend AT %Q* : BOOL;	
	//NOT USED BUT USABLE	
	DI_BoundaryPressure AT %I* : BOOL;
END_VAR

                  
                

ACTION ACT_Extend:
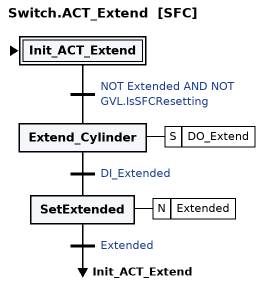
INITIAL_STEP Init_ACT_Extend:
END_STEP
TRANSITION FROM Init_ACT_Extend TO Extend_Cylinder
  := NOT Extended AND NOT GVL.IsSFCResetting;
END_TRANSITION
STEP Extend_Cylinder:
  DO_Extend(S);
END_STEP
TRANSITION FROM Extend_Cylinder TO SetExtended
  := DI_Extended;
END_TRANSITION
STEP SetExtended:
  Extended(N);
END_STEP
TRANSITION FROM SetExtended TO Init_ACT_Extend
  := Extended;
END_TRANSITION
END_ACTION

ACTION ACT_Retract:
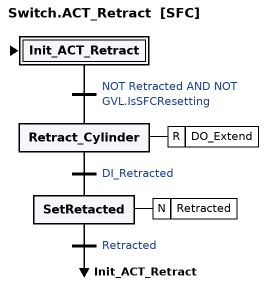
INITIAL_STEP Init_ACT_Retract:
END_STEP
TRANSITION FROM Init_ACT_Retract TO Retract_Cylinder
  := NOT Retracted AND NOT GVL.IsSFCResetting;
END_TRANSITION
STEP Retract_Cylinder:
  DO_Extend(R);
END_STEP
TRANSITION FROM Retract_Cylinder TO SetRetacted
  := DI_Retracted;
END_TRANSITION
STEP SetRetacted:
  Retracted(N);
END_STEP
TRANSITION FROM SetRetacted TO Init_ACT_Retract
  := Retracted;
END_TRANSITION
END_ACTION
END_FUNCTION_BLOCK

FUNCTION_BLOCK TurningTable
VAR_INPUT
END_VAR
VAR_OUTPUT
	//Hardware
	Motor : Motor;
	AtStack : MicroSwitch;
	AtConveyor : MicroSwitch;
	AtStamp : MicroSwitch;
	Potentiometer : Potentiometer;
END_VAR
VAR	
	//NOT USED BUT USABLE
	AtStackInd : InductiveSwitch;
	BetweenStackConveyor : InductiveSwitch;
	AtConveyorInd : InductiveSwitch;
	BetweenConveyorStamp : InductiveSwitch;
	AtStampInd : InductiveSwitch;

END_VAR

                  Potentiometer();
                
END_FUNCTION_BLOCK

FUNCTION_BLOCK UltrasonicSensor
VAR_INPUT
END_VAR
VAR_OUTPUT
END_VAR
VAR
	AI_UltraSonic AT %I* : INT;
END_VAR

                  
                
END_FUNCTION_BLOCK

FUNCTION_BLOCK VacuumGripper
VAR_INPUT	
	//Hardware
	Valve : Valve;
	VacuumSwitch : VacuumSwitch;
END_VAR
VAR_OUTPUT	
	//Software
	Intaken : BOOL;
	Released : BOOL;
END_VAR
VAR	
	//NOT USED BUT USABLE
	AI_VacuumSensor AT %I* : INT;	
	DI_BoundaryVacuumPressure AT %I* : BOOL;
	DI_VacuumBoundaryFlowPressure1 AT %I* : BOOL;
	DI_VacuumBoundaryFlowPressure2 AT %I* : BOOL;	
	AI_VacuumPressure AT %I* : INT;
END_VAR

                  
                

ACTION ACT_Intake:
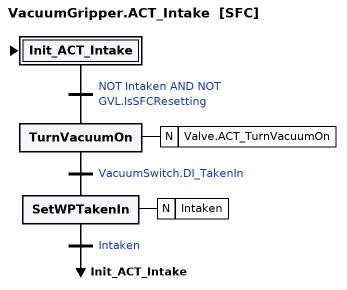
INITIAL_STEP Init_ACT_Intake:
END_STEP
TRANSITION FROM Init_ACT_Intake TO TurnVacuumOn
  := NOT Intaken AND NOT GVL.IsSFCResetting;
END_TRANSITION
STEP TurnVacuumOn:
  Valve.ACT_TurnVacuumOn(N);
END_STEP
TRANSITION FROM TurnVacuumOn TO SetWPTakenIn
  := VacuumSwitch.DI_TakenIn;
END_TRANSITION
STEP SetWPTakenIn:
  Intaken(N);
END_STEP
TRANSITION FROM SetWPTakenIn TO Init_ACT_Intake
  := Intaken;
END_TRANSITION
END_ACTION

ACTION ACT_Release:
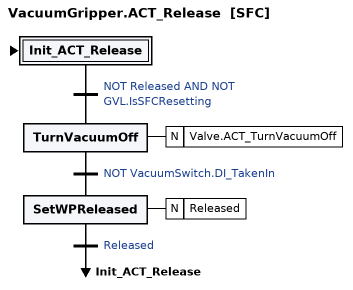
INITIAL_STEP Init_ACT_Release:
END_STEP
TRANSITION FROM Init_ACT_Release TO TurnVacuumOff
  := NOT Released AND NOT GVL.IsSFCResetting;
END_TRANSITION
STEP TurnVacuumOff:
  Valve.ACT_TurnVacuumOff(N);
END_STEP
TRANSITION FROM TurnVacuumOff TO SetWPReleased
  := NOT VacuumSwitch.DI_TakenIn;
END_TRANSITION
STEP SetWPReleased:
  Released(N);
END_STEP
TRANSITION FROM SetWPReleased TO Init_ACT_Release
  := Released;
END_TRANSITION
END_ACTION
END_FUNCTION_BLOCK

FUNCTION_BLOCK VacuumGripperExtended
VAR_INPUT	
	//Hardware
	Valve : Valve;
	VacuumSwitch : VacuumSwitch;
END_VAR
VAR_OUTPUT	
	//Software
	Intaken : BOOL;
	Released : BOOL;
END_VAR
VAR	
	//Hardware
	VacuumHit AT %Q* : BOOL;
	//NOT USED BUT USABLE
	AI_VacuumSensor AT %I* : INT;
	DI_BoundaryVacuumPressure AT %I* : BOOL;
	DI_VacuumBoundaryFlowPressure1 AT %I* : BOOL;
	DI_VacuumBoundaryFlowPressure2 AT %I* : BOOL;	
	AI_VacuumPressure AT %I* : INT;
END_VAR

                  
                

ACTION ACT_Intake:
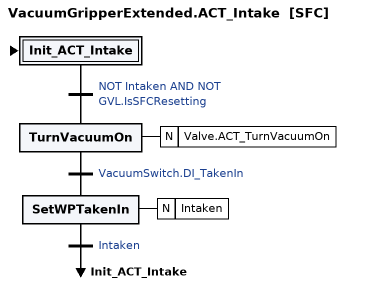
INITIAL_STEP Init_ACT_Intake:
END_STEP
TRANSITION FROM Init_ACT_Intake TO TurnVacuumOn
  := NOT Intaken AND NOT GVL.IsSFCResetting;
END_TRANSITION
STEP TurnVacuumOn:
  Valve.ACT_TurnVacuumOn(N);
END_STEP
TRANSITION FROM TurnVacuumOn TO SetWPTakenIn
  := VacuumSwitch.DI_TakenIn;
END_TRANSITION
STEP SetWPTakenIn:
  Intaken(N);
END_STEP
TRANSITION FROM SetWPTakenIn TO Init_ACT_Intake
  := Intaken;
END_TRANSITION
END_ACTION

ACTION ACT_Release:
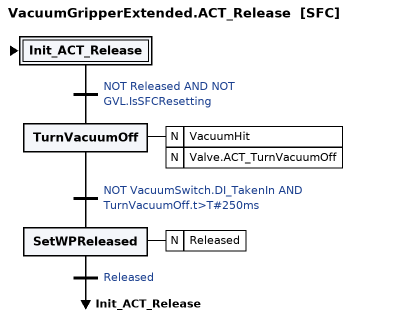
INITIAL_STEP Init_ACT_Release:
END_STEP
TRANSITION FROM Init_ACT_Release TO TurnVacuumOff
  := NOT Released AND NOT GVL.IsSFCResetting;
END_TRANSITION
STEP TurnVacuumOff:
  VacuumHit(N);
  Valve.ACT_TurnVacuumOff(N);
END_STEP
TRANSITION FROM TurnVacuumOff TO SetWPReleased
  := NOT VacuumSwitch.DI_TakenIn AND TurnVacuumOff.t>T#250ms;
END_TRANSITION
STEP SetWPReleased:
  Released(N);
END_STEP
TRANSITION FROM SetWPReleased TO Init_ACT_Release
  := Released;
END_TRANSITION
END_ACTION
END_FUNCTION_BLOCK

FUNCTION_BLOCK VacuumSwitch
VAR_INPUT
END_VAR
VAR_OUTPUT
	//Hardware
	DI_TakenIn AT %I* : BOOL;
END_VAR
VAR
END_VAR

                  
                
END_FUNCTION_BLOCK

FUNCTION_BLOCK Valve
VAR_INPUT
END_VAR
VAR_OUTPUT
END_VAR
VAR	
	//Hardware
	DO_VacuumOn AT %Q* : BOOL;
END_VAR

                  
                

ACTION ACT_TurnVacuumOff:
                      DO_VacuumOn := FALSE;
                    
END_ACTION

ACTION ACT_TurnVacuumOn:
                      DO_VacuumOn := TRUE;
                    
END_ACTION
END_FUNCTION_BLOCK

FUNCTION_BLOCK ValveBlock
VAR_INPUT
END_VAR
VAR_OUTPUT
END_VAR
VAR
	DI_BoundaryPressure AT %I* : BOOL; 
	DI_BoundaryFlowPressure AT %I* : BOOL; 
	AI_PressureSensor AT %I* : INT; 
	AI_FlowPressure AT %I* : INT; 
	DO_SetBlockPressure AT %Q* : BOOL;
END_VAR

                  
                

ACTION ACT_BlockadeBlockPressure:
                      DO_SetBlockPressure := TRUE;
                    
END_ACTION

ACTION ACT_ReleaseBlockPressure:
                      DO_SetBlockPressure := FALSE;
                    
END_ACTION
END_FUNCTION_BLOCK

FUNCTION_BLOCK WeightModule
VAR_INPUT
END_VAR
VAR_OUTPUT
END_VAR
VAR
	AI_WPWeight AT %I* : INT;
END_VAR

                  
                
END_FUNCTION_BLOCK

FUNCTION_BLOCK Crane
VAR_INPUT
	bSR : BOOL;
	bCR : BOOL;
	bStR : BOOL;

	//Hardware
	LiftingCylinder : MonostableCylinder;
	Gripper : VacuumGripper;	
	Table : TurningTable;		
	RFID : RFID;
	
	//Software		
	SoftwareEmergency : BOOL;	
	Check_Stack_WPProvided : BOOL;
	Check_Stack_WPType_Black : BOOL;
	Check_Stack_WPType_White : BOOL;
	Check_Stack_WPType_Metallic : BOOL;
	Check_LargeSortingConveyor_IsSorting : BOOL;
	Check_LargeSortingConveyor_AutomaticExecuteCompleted : BOOL;	
	Check_Stamp_IsStamping : BOOL;
	Check_Stamp_WPAvailable : BOOL;
	Check_Stamp_AutomaticExecuteCompleted : BOOL;
	Check_RefillConveyor_IsSending : BOOL;
	Check_EngineStop : BOOL;
	SFCReset : BOOL;	//Only for SFC implementation
END_VAR
VAR_OUTPUT	
	//Software
	InitCompleted : BOOL;
	AutomaticExecuteCompleted : BOOL;			
	Conveyor_AllowedToOperate : BOOL;
	Stamp_AllowedToOperate : BOOL;	
	WPPickedUp : BOOL;
	EmergencyHandled : BOOL;	
END_VAR
VAR		
	//Hardware		
	CraneSpeed AT %Q* : INT;
	
	//Software
	WPPutDown : BOOL;
	ReachedStack : BOOL;
	ReachedStackRFID : BOOL;
	ReachedConveyor : BOOL;
	ReachedConveyorRFID : BOOL;
	ReachedStamp : BOOL;	
	ReachedStampRFID : BOOL;
	WPType_White : BOOL;
	WPType_Black : BOOL;
	WPType_Metallic : BOOL;
	WPWeight_Light : BOOL;
	WPWeight_Medium : BOOL;
	WPWeight_Heavy : BOOL;
END_VAR

                  Table();
Check_Stack_WPProvided := Main.Stack_WPProvided;
Check_Stack_WPType_Black := Main.Stack_WPType_Black;
Check_Stack_WPType_White := Main.Stack_WPType_White;
Check_Stack_WPType_Metallic := Main.Stack_WPType_Metallic;
Check_LargeSortingConveyor_IsSorting := Main.LargeSortingConveyor_IsSorting;
Check_LargeSortingConveyor_AutomaticExecuteCompleted := Main.LargeSortingConveyor_AutomaticExecuteCompleted;
Check_Stamp_IsStamping := Main.Stamp_IsStamping;
Check_Stamp_WPAvailable := Main.Stamp_WPAvailable;
Check_Stamp_AutomaticExecuteCompleted := Main.Stamp_AutomaticExecuteCompleted;
Check_RefillConveyor_IsSending := Main.Check_RefillConveyor_IsSending;
Check_EngineStop := MAIN.PPU_EngineStop;
IF Check_EngineStop THEN
	Table.Motor.ACT_Stop();
END_IF

IF(bSR AND NOT ReachedStackRFID)THEN
	ACT_MoveToStackRFID();
END_IF
IF(bCR AND NOT ReachedConveyorRFID)THEN
	ACT_MoveToConveyorRFID();
END_IF
IF(bStR AND NOT ReachedStampRFID)THEN
	ACT_MoveToStampRFID();
END_IF
                

ACTION Reset_ConveyorAllowedToOperate:
                      Conveyor_AllowedToOperate := FALSE;
                    
END_ACTION

ACTION Reset_StampAllowedToOperate:
                      Stamp_AllowedToOperate := FALSE;
                    
END_ACTION

ACTION Reset_Variables:
                      InitCompleted := FALSE;
AutomaticExecuteCompleted := FALSE;
Conveyor_AllowedToOperate := FALSE;
Stamp_AllowedToOperate := FALSE;

WPPickedUp := FALSE;
WPPutDown := FALSE;
ReachedStack := FALSE;
ReachedConveyor := FALSE;
ReachedStamp := FALSE;	
WPType_White := FALSE;
WPType_Black := FALSE;
WPType_Metallic := FALSE;
WPWeight_Light := FALSE;
WPWeight_Medium := FALSE;
WPWeight_Heavy := FALSE;
                    
END_ACTION

ACTION Set_ConveyorAllowedToOperate:
                      Conveyor_AllowedToOperate := TRUE;
                    
END_ACTION

ACTION Set_StampAllowedToOperate:
                      Stamp_AllowedToOperate := TRUE;
                    
END_ACTION

ACTION Set_WPTypeEqualsStack:
                      WPType_White:=Main.Stack_WPType_White;
WPType_Black:=Main.Stack_WPType_Black;	
WPType_Metallic:=Main.Stack_WPType_Metallic;
WPWeight_Light:=Main.Stack_WPWeight_Light;
WPWeight_Medium:=Main.Stack_WPWeight_Medium;	
WPWeight_Heavy:=Main.Stack_WPWeight_Heavy;
                    
END_ACTION

ACTION Set_WPTypeEqualsStamp:
                      WPType_White:=Main.Stamp_WPType_White;
WPType_Black:=Main.Stamp_WPType_Black;	
WPType_Metallic:=Main.Stamp_WPType_Metallic;
WPWeight_Light:=Main.Stamp_WPWeight_Light;
WPWeight_Medium:=Main.Stamp_WPWeight_Medium;	
WPWeight_Heavy:=Main.Stamp_WPWeight_Heavy;
                    
END_ACTION

ACTION ACT_MoveToConveyor:
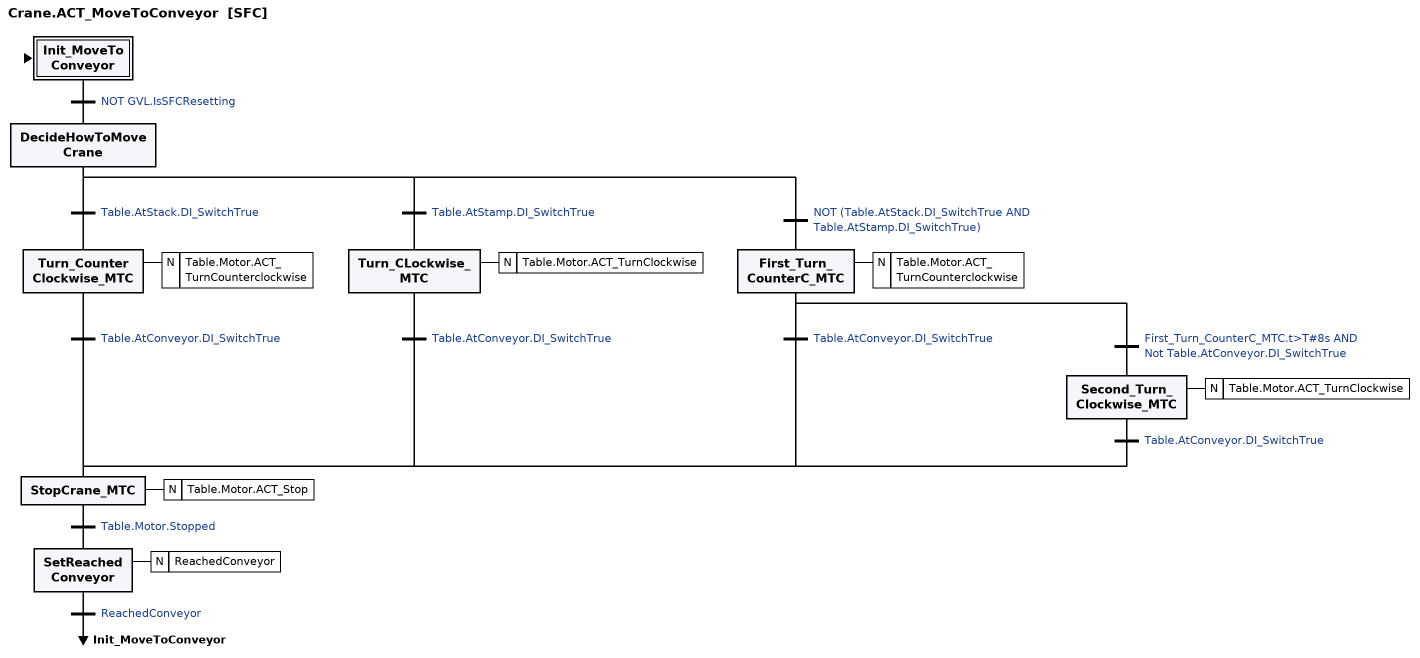
INITIAL_STEP Init_MoveToConveyor:
END_STEP
TRANSITION FROM Init_MoveToConveyor TO DecideHowToMoveCrane
  := NOT GVL.IsSFCResetting;
END_TRANSITION
STEP DecideHowToMoveCrane:
END_STEP
TRANSITION FROM DecideHowToMoveCrane TO Turn_CounterClockwise_MTC
  := Table.AtStack.DI_SwitchTrue;
END_TRANSITION
TRANSITION FROM DecideHowToMoveCrane TO Turn_CLockwise_MTC
  := Table.AtStamp.DI_SwitchTrue;
END_TRANSITION
TRANSITION FROM DecideHowToMoveCrane TO First_Turn_CounterC_MTC
  := NOT (Table.AtStack.DI_SwitchTrue AND Table.AtStamp.DI_SwitchTrue);
END_TRANSITION
STEP Turn_CounterClockwise_MTC:
  Table.Motor.ACT_TurnCounterclockwise(N);
END_STEP
TRANSITION FROM Turn_CounterClockwise_MTC TO StopCrane_MTC
  := Table.AtConveyor.DI_SwitchTrue;
END_TRANSITION
STEP Turn_CLockwise_MTC:
  Table.Motor.ACT_TurnClockwise(N);
END_STEP
TRANSITION FROM Turn_CLockwise_MTC TO StopCrane_MTC
  := Table.AtConveyor.DI_SwitchTrue;
END_TRANSITION
STEP First_Turn_CounterC_MTC:
  Table.Motor.ACT_TurnCounterclockwise(N);
END_STEP
TRANSITION FROM First_Turn_CounterC_MTC TO StopCrane_MTC
  := Table.AtConveyor.DI_SwitchTrue;
END_TRANSITION
TRANSITION FROM First_Turn_CounterC_MTC TO Second_Turn_Clockwise_MTC
  := First_Turn_CounterC_MTC.t>T#8s AND Not Table.AtConveyor.DI_SwitchTrue;
END_TRANSITION
STEP Second_Turn_Clockwise_MTC:
  Table.Motor.ACT_TurnClockwise(N);
END_STEP
TRANSITION FROM Second_Turn_Clockwise_MTC TO StopCrane_MTC
  := Table.AtConveyor.DI_SwitchTrue;
END_TRANSITION
STEP StopCrane_MTC:
  Table.Motor.ACT_Stop(N);
END_STEP
TRANSITION FROM StopCrane_MTC TO SetReachedConveyor
  := Table.Motor.Stopped;
END_TRANSITION
STEP SetReachedConveyor:
  ReachedConveyor(N);
END_STEP
TRANSITION FROM SetReachedConveyor TO Init_MoveToConveyor
  := ReachedConveyor;
END_TRANSITION
END_ACTION

ACTION ACT_MoveToConveyorRFID:
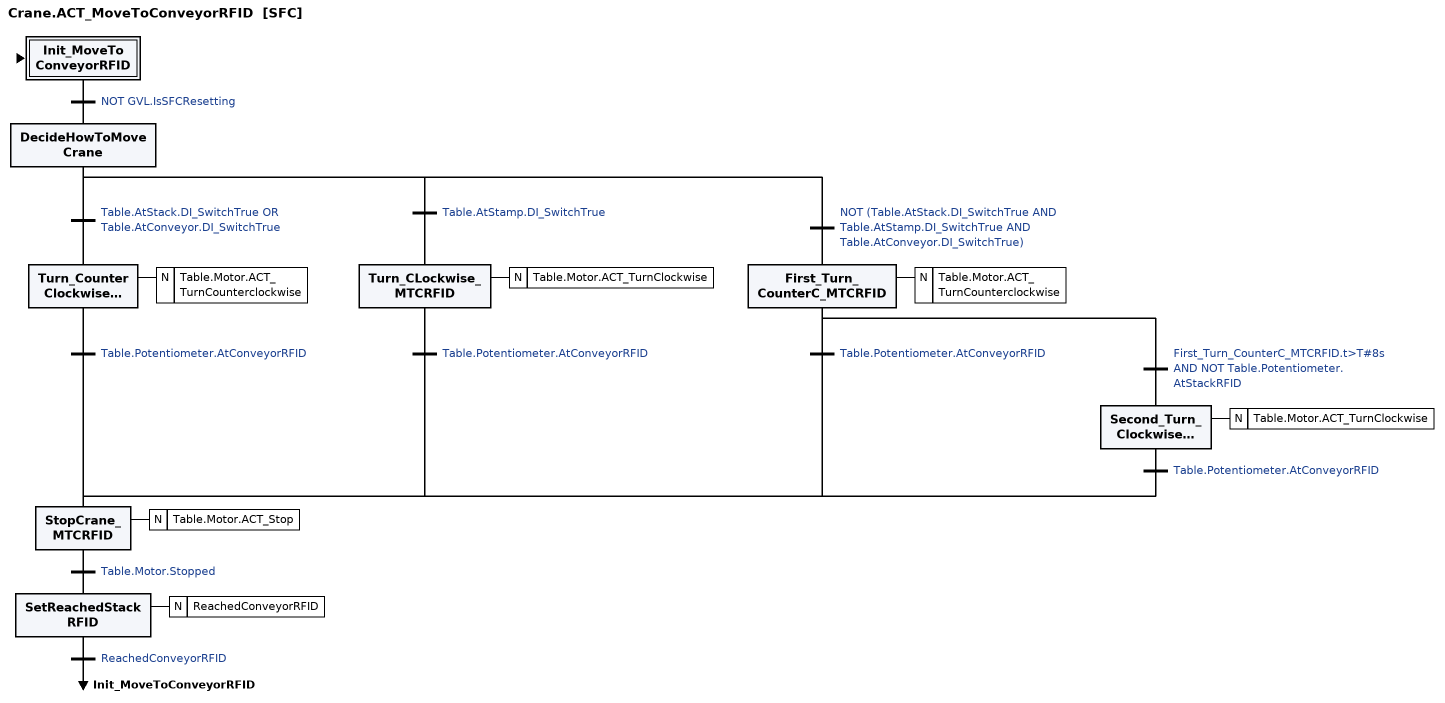
INITIAL_STEP Init_MoveToConveyorRFID:
END_STEP
TRANSITION FROM Init_MoveToConveyorRFID TO DecideHowToMoveCrane
  := NOT GVL.IsSFCResetting;
END_TRANSITION
STEP DecideHowToMoveCrane:
END_STEP
TRANSITION FROM DecideHowToMoveCrane TO Turn_CounterClockwise_MTCRFID
  := Table.AtStack.DI_SwitchTrue OR Table.AtConveyor.DI_SwitchTrue;
END_TRANSITION
TRANSITION FROM DecideHowToMoveCrane TO Turn_CLockwise_MTCRFID
  := Table.AtStamp.DI_SwitchTrue;
END_TRANSITION
TRANSITION FROM DecideHowToMoveCrane TO First_Turn_CounterC_MTCRFID
  := NOT (Table.AtStack.DI_SwitchTrue AND Table.AtStamp.DI_SwitchTrue AND Table.AtConveyor.DI_SwitchTrue);
END_TRANSITION
STEP Turn_CounterClockwise_MTCRFID:
  Table.Motor.ACT_TurnCounterclockwise(N);
END_STEP
TRANSITION FROM Turn_CounterClockwise_MTCRFID TO StopCrane_MTCRFID
  := Table.Potentiometer.AtConveyorRFID;
END_TRANSITION
STEP Turn_CLockwise_MTCRFID:
  Table.Motor.ACT_TurnClockwise(N);
END_STEP
TRANSITION FROM Turn_CLockwise_MTCRFID TO StopCrane_MTCRFID
  := Table.Potentiometer.AtConveyorRFID;
END_TRANSITION
STEP First_Turn_CounterC_MTCRFID:
  Table.Motor.ACT_TurnCounterclockwise(N);
END_STEP
TRANSITION FROM First_Turn_CounterC_MTCRFID TO StopCrane_MTCRFID
  := Table.Potentiometer.AtConveyorRFID;
END_TRANSITION
TRANSITION FROM First_Turn_CounterC_MTCRFID TO Second_Turn_Clockwise_MTCRFID
  := First_Turn_CounterC_MTCRFID.t>T#8s AND NOT Table.Potentiometer.AtStackRFID;
END_TRANSITION
STEP Second_Turn_Clockwise_MTCRFID:
  Table.Motor.ACT_TurnClockwise(N);
END_STEP
TRANSITION FROM Second_Turn_Clockwise_MTCRFID TO StopCrane_MTCRFID
  := Table.Potentiometer.AtConveyorRFID;
END_TRANSITION
STEP StopCrane_MTCRFID:
  Table.Motor.ACT_Stop(N);
END_STEP
TRANSITION FROM StopCrane_MTCRFID TO SetReachedStackRFID
  := Table.Motor.Stopped;
END_TRANSITION
STEP SetReachedStackRFID:
  ReachedConveyorRFID(N);
END_STEP
TRANSITION FROM SetReachedStackRFID TO Init_MoveToConveyorRFID
  := ReachedConveyorRFID;
END_TRANSITION
END_ACTION

ACTION ACT_MoveToStack:
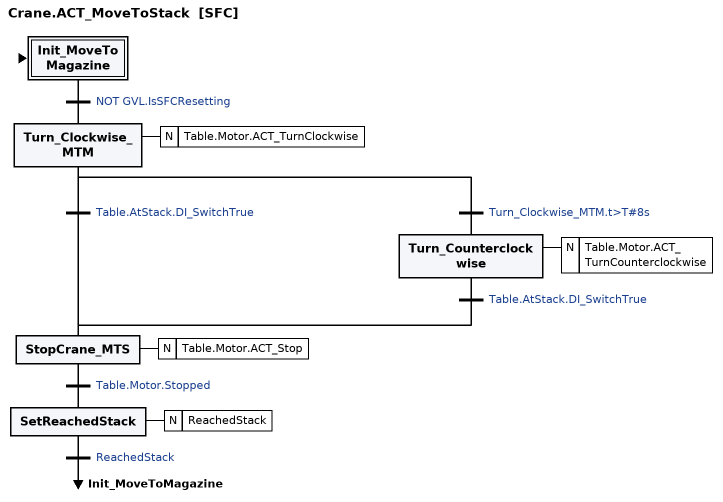
INITIAL_STEP Init_MoveToMagazine:
END_STEP
TRANSITION FROM Init_MoveToMagazine TO Turn_Clockwise_MTM
  := NOT GVL.IsSFCResetting;
END_TRANSITION
STEP Turn_Clockwise_MTM:
  Table.Motor.ACT_TurnClockwise(N);
END_STEP
TRANSITION FROM Turn_Clockwise_MTM TO StopCrane_MTS
  := Table.AtStack.DI_SwitchTrue;
END_TRANSITION
TRANSITION FROM Turn_Clockwise_MTM TO Turn_Counterclockwise
  := Turn_Clockwise_MTM.t>T#8s;
END_TRANSITION
STEP Turn_Counterclockwise:
  Table.Motor.ACT_TurnCounterclockwise(N);
END_STEP
TRANSITION FROM Turn_Counterclockwise TO StopCrane_MTS
  := Table.AtStack.DI_SwitchTrue;
END_TRANSITION
STEP StopCrane_MTS:
  Table.Motor.ACT_Stop(N);
END_STEP
TRANSITION FROM StopCrane_MTS TO SetReachedStack
  := Table.Motor.Stopped;
END_TRANSITION
STEP SetReachedStack:
  ReachedStack(N);
END_STEP
TRANSITION FROM SetReachedStack TO Init_MoveToMagazine
  := ReachedStack;
END_TRANSITION
END_ACTION

ACTION ACT_MoveToStackRFID:
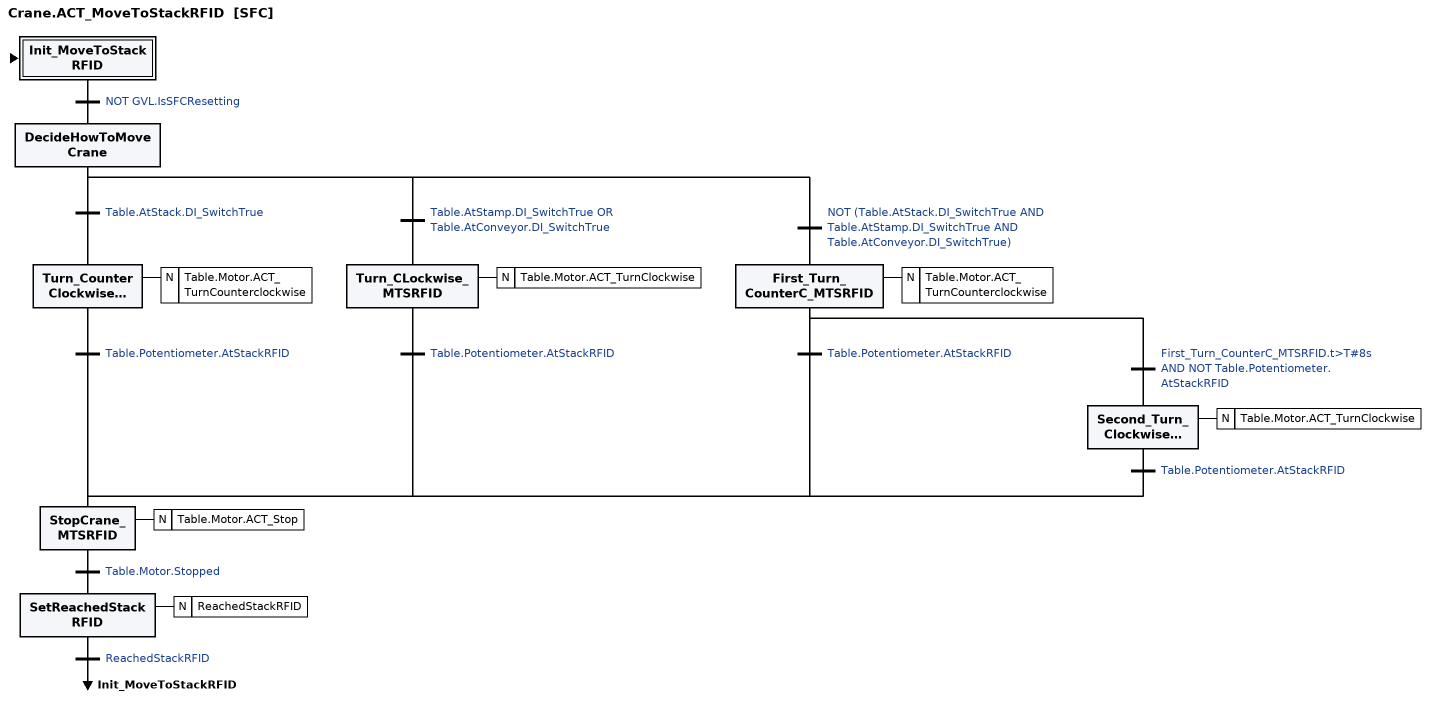
INITIAL_STEP Init_MoveToStackRFID:
END_STEP
TRANSITION FROM Init_MoveToStackRFID TO DecideHowToMoveCrane
  := NOT GVL.IsSFCResetting;
END_TRANSITION
STEP DecideHowToMoveCrane:
END_STEP
TRANSITION FROM DecideHowToMoveCrane TO Turn_CounterClockwise_MTSRFID
  := Table.AtStack.DI_SwitchTrue;
END_TRANSITION
TRANSITION FROM DecideHowToMoveCrane TO Turn_CLockwise_MTSRFID
  := Table.AtStamp.DI_SwitchTrue OR Table.AtConveyor.DI_SwitchTrue;
END_TRANSITION
TRANSITION FROM DecideHowToMoveCrane TO First_Turn_CounterC_MTSRFID
  := NOT (Table.AtStack.DI_SwitchTrue AND Table.AtStamp.DI_SwitchTrue AND Table.AtConveyor.DI_SwitchTrue);
END_TRANSITION
STEP Turn_CounterClockwise_MTSRFID:
  Table.Motor.ACT_TurnCounterclockwise(N);
END_STEP
TRANSITION FROM Turn_CounterClockwise_MTSRFID TO StopCrane_MTSRFID
  := Table.Potentiometer.AtStackRFID;
END_TRANSITION
STEP Turn_CLockwise_MTSRFID:
  Table.Motor.ACT_TurnClockwise(N);
END_STEP
TRANSITION FROM Turn_CLockwise_MTSRFID TO StopCrane_MTSRFID
  := Table.Potentiometer.AtStackRFID;
END_TRANSITION
STEP First_Turn_CounterC_MTSRFID:
  Table.Motor.ACT_TurnCounterclockwise(N);
END_STEP
TRANSITION FROM First_Turn_CounterC_MTSRFID TO StopCrane_MTSRFID
  := Table.Potentiometer.AtStackRFID;
END_TRANSITION
TRANSITION FROM First_Turn_CounterC_MTSRFID TO Second_Turn_Clockwise_MTSRFID
  := First_Turn_CounterC_MTSRFID.t>T#8s AND NOT Table.Potentiometer.AtStackRFID;
END_TRANSITION
STEP Second_Turn_Clockwise_MTSRFID:
  Table.Motor.ACT_TurnClockwise(N);
END_STEP
TRANSITION FROM Second_Turn_Clockwise_MTSRFID TO StopCrane_MTSRFID
  := Table.Potentiometer.AtStackRFID;
END_TRANSITION
STEP StopCrane_MTSRFID:
  Table.Motor.ACT_Stop(N);
END_STEP
TRANSITION FROM StopCrane_MTSRFID TO SetReachedStackRFID
  := Table.Motor.Stopped;
END_TRANSITION
STEP SetReachedStackRFID:
  ReachedStackRFID(N);
END_STEP
TRANSITION FROM SetReachedStackRFID TO Init_MoveToStackRFID
  := ReachedStackRFID;
END_TRANSITION
END_ACTION

ACTION ACT_MoveToStamp:
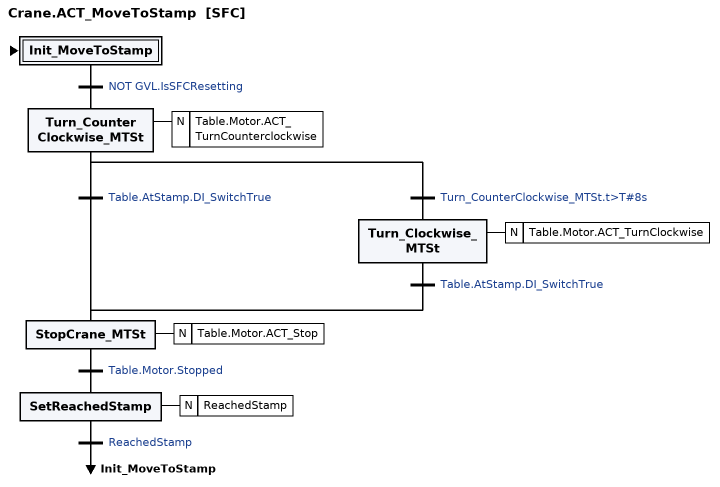
INITIAL_STEP Init_MoveToStamp:
END_STEP
TRANSITION FROM Init_MoveToStamp TO Turn_CounterClockwise_MTSt
  := NOT GVL.IsSFCResetting;
END_TRANSITION
STEP Turn_CounterClockwise_MTSt:
  Table.Motor.ACT_TurnCounterclockwise(N);
END_STEP
TRANSITION FROM Turn_CounterClockwise_MTSt TO StopCrane_MTSt
  := Table.AtStamp.DI_SwitchTrue;
END_TRANSITION
TRANSITION FROM Turn_CounterClockwise_MTSt TO Turn_Clockwise_MTSt
  := Turn_CounterClockwise_MTSt.t>T#8s;
END_TRANSITION
STEP Turn_Clockwise_MTSt:
  Table.Motor.ACT_TurnClockwise(N);
END_STEP
TRANSITION FROM Turn_Clockwise_MTSt TO StopCrane_MTSt
  := Table.AtStamp.DI_SwitchTrue;
END_TRANSITION
STEP StopCrane_MTSt:
  Table.Motor.ACT_Stop(N);
END_STEP
TRANSITION FROM StopCrane_MTSt TO SetReachedStamp
  := Table.Motor.Stopped;
END_TRANSITION
STEP SetReachedStamp:
  ReachedStamp(N);
END_STEP
TRANSITION FROM SetReachedStamp TO Init_MoveToStamp
  := ReachedStamp;
END_TRANSITION
END_ACTION

ACTION ACT_MoveToStampRFID:
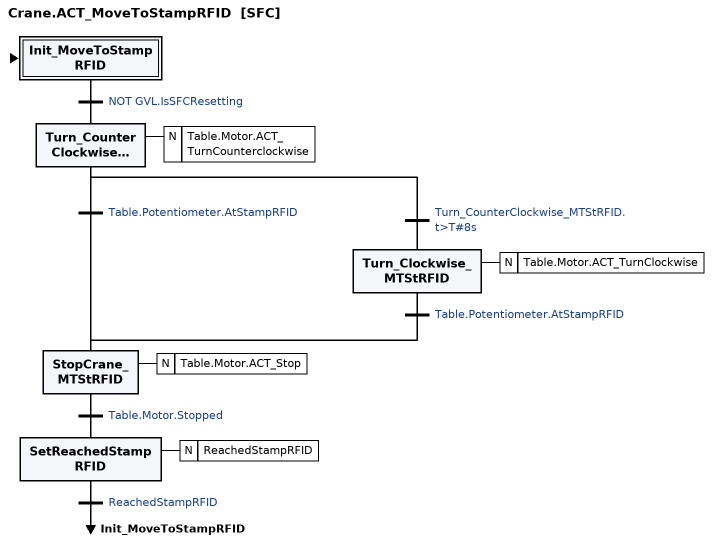
INITIAL_STEP Init_MoveToStampRFID:
END_STEP
TRANSITION FROM Init_MoveToStampRFID TO Turn_CounterClockwise_MTStRFID
  := NOT GVL.IsSFCResetting;
END_TRANSITION
STEP Turn_CounterClockwise_MTStRFID:
  Table.Motor.ACT_TurnCounterclockwise(N);
END_STEP
TRANSITION FROM Turn_CounterClockwise_MTStRFID TO StopCrane_MTStRFID
  := Table.Potentiometer.AtStampRFID;
END_TRANSITION
TRANSITION FROM Turn_CounterClockwise_MTStRFID TO Turn_Clockwise_MTStRFID
  := Turn_CounterClockwise_MTStRFID.t>T#8s;
END_TRANSITION
STEP Turn_Clockwise_MTStRFID:
  Table.Motor.ACT_TurnClockwise(N);
END_STEP
TRANSITION FROM Turn_Clockwise_MTStRFID TO StopCrane_MTStRFID
  := Table.Potentiometer.AtStampRFID;
END_TRANSITION
STEP StopCrane_MTStRFID:
  Table.Motor.ACT_Stop(N);
END_STEP
TRANSITION FROM StopCrane_MTStRFID TO SetReachedStampRFID
  := Table.Motor.Stopped;
END_TRANSITION
STEP SetReachedStampRFID:
  ReachedStampRFID(N);
END_STEP
TRANSITION FROM SetReachedStampRFID TO Init_MoveToStampRFID
  := ReachedStampRFID;
END_TRANSITION
END_ACTION

ACTION ACT_PickUpWP:
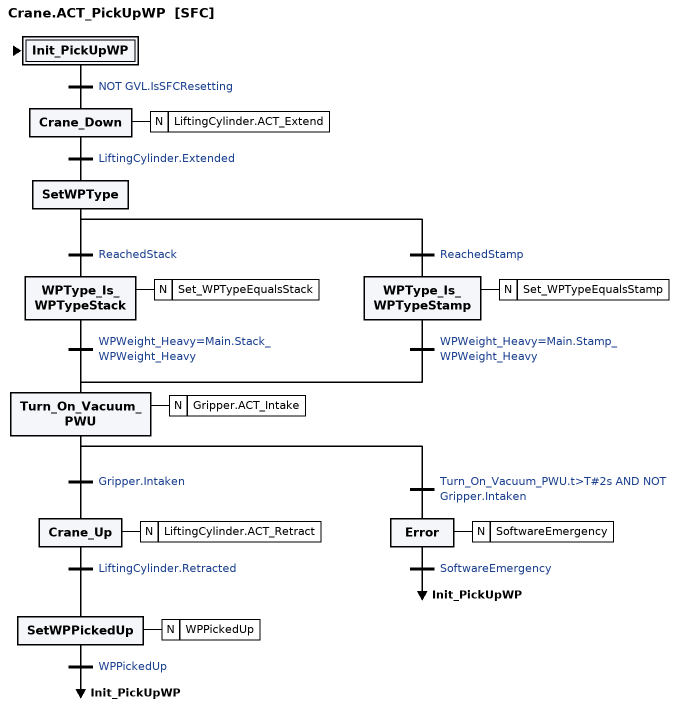
INITIAL_STEP Init_PickUpWP:
END_STEP
TRANSITION FROM Init_PickUpWP TO Crane_Down
  := NOT GVL.IsSFCResetting;
END_TRANSITION
STEP Crane_Down:
  LiftingCylinder.ACT_Extend(N);
END_STEP
TRANSITION FROM Crane_Down TO SetWPType
  := LiftingCylinder.Extended;
END_TRANSITION
STEP SetWPType:
END_STEP
TRANSITION FROM SetWPType TO WPType_Is_WPTypeStack
  := ReachedStack;
END_TRANSITION
TRANSITION FROM SetWPType TO WPType_Is_WPTypeStamp
  := ReachedStamp;
END_TRANSITION
STEP WPType_Is_WPTypeStack:
  Set_WPTypeEqualsStack(N);
END_STEP
TRANSITION FROM WPType_Is_WPTypeStack TO Turn_On_Vacuum_PWU
  := WPWeight_Heavy=Main.Stack_WPWeight_Heavy;
END_TRANSITION
STEP WPType_Is_WPTypeStamp:
  Set_WPTypeEqualsStamp(N);
END_STEP
TRANSITION FROM WPType_Is_WPTypeStamp TO Turn_On_Vacuum_PWU
  := WPWeight_Heavy=Main.Stamp_WPWeight_Heavy;
END_TRANSITION
STEP Turn_On_Vacuum_PWU:
  Gripper.ACT_Intake(N);
END_STEP
TRANSITION FROM Turn_On_Vacuum_PWU TO Crane_Up
  := Gripper.Intaken;
END_TRANSITION
TRANSITION FROM Turn_On_Vacuum_PWU TO Error
  := Turn_On_Vacuum_PWU.t>T#2s AND NOT Gripper.Intaken;
END_TRANSITION
STEP Crane_Up:
  LiftingCylinder.ACT_Retract(N);
END_STEP
TRANSITION FROM Crane_Up TO SetWPPickedUp
  := LiftingCylinder.Retracted;
END_TRANSITION
STEP Error:
  SoftwareEmergency(N);
END_STEP
TRANSITION FROM Error TO Init_PickUpWP
  := SoftwareEmergency;
END_TRANSITION
STEP SetWPPickedUp:
  WPPickedUp(N);
END_STEP
TRANSITION FROM SetWPPickedUp TO Init_PickUpWP
  := WPPickedUp;
END_TRANSITION
END_ACTION

ACTION ACT_PutDownWP:
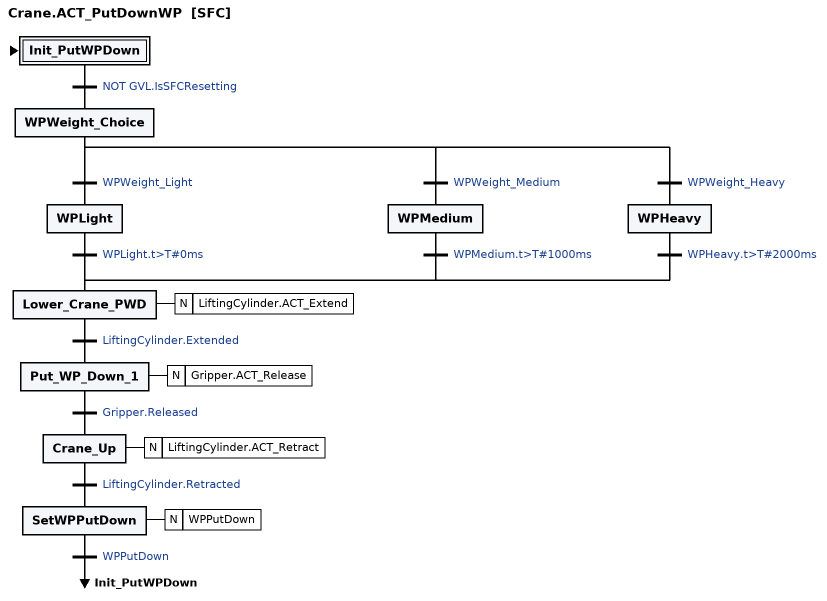
INITIAL_STEP Init_PutWPDown:
END_STEP
TRANSITION FROM Init_PutWPDown TO WPWeight_Choice
  := NOT GVL.IsSFCResetting;
END_TRANSITION
STEP WPWeight_Choice:
END_STEP
TRANSITION FROM WPWeight_Choice TO WPLight
  := WPWeight_Light;
END_TRANSITION
TRANSITION FROM WPWeight_Choice TO WPMedium
  := WPWeight_Medium;
END_TRANSITION
TRANSITION FROM WPWeight_Choice TO WPHeavy
  := WPWeight_Heavy;
END_TRANSITION
STEP WPLight:
END_STEP
TRANSITION FROM WPLight TO Lower_Crane_PWD
  := WPLight.t>T#0ms;
END_TRANSITION
STEP WPMedium:
END_STEP
TRANSITION FROM WPMedium TO Lower_Crane_PWD
  := WPMedium.t>T#1000ms;
END_TRANSITION
STEP WPHeavy:
END_STEP
TRANSITION FROM WPHeavy TO Lower_Crane_PWD
  := WPHeavy.t>T#2000ms;
END_TRANSITION
STEP Lower_Crane_PWD:
  LiftingCylinder.ACT_Extend(N);
END_STEP
TRANSITION FROM Lower_Crane_PWD TO Put_WP_Down_1
  := LiftingCylinder.Extended;
END_TRANSITION
STEP Put_WP_Down_1:
  Gripper.ACT_Release(N);
END_STEP
TRANSITION FROM Put_WP_Down_1 TO Crane_Up
  := Gripper.Released;
END_TRANSITION
STEP Crane_Up:
  LiftingCylinder.ACT_Retract(N);
END_STEP
TRANSITION FROM Crane_Up TO SetWPPutDown
  := LiftingCylinder.Retracted;
END_TRANSITION
STEP SetWPPutDown:
  WPPutDown(N);
END_STEP
TRANSITION FROM SetWPPutDown TO Init_PutWPDown
  := WPPutDown;
END_TRANSITION
END_ACTION

ACTION ACT_AutomaticExecute:
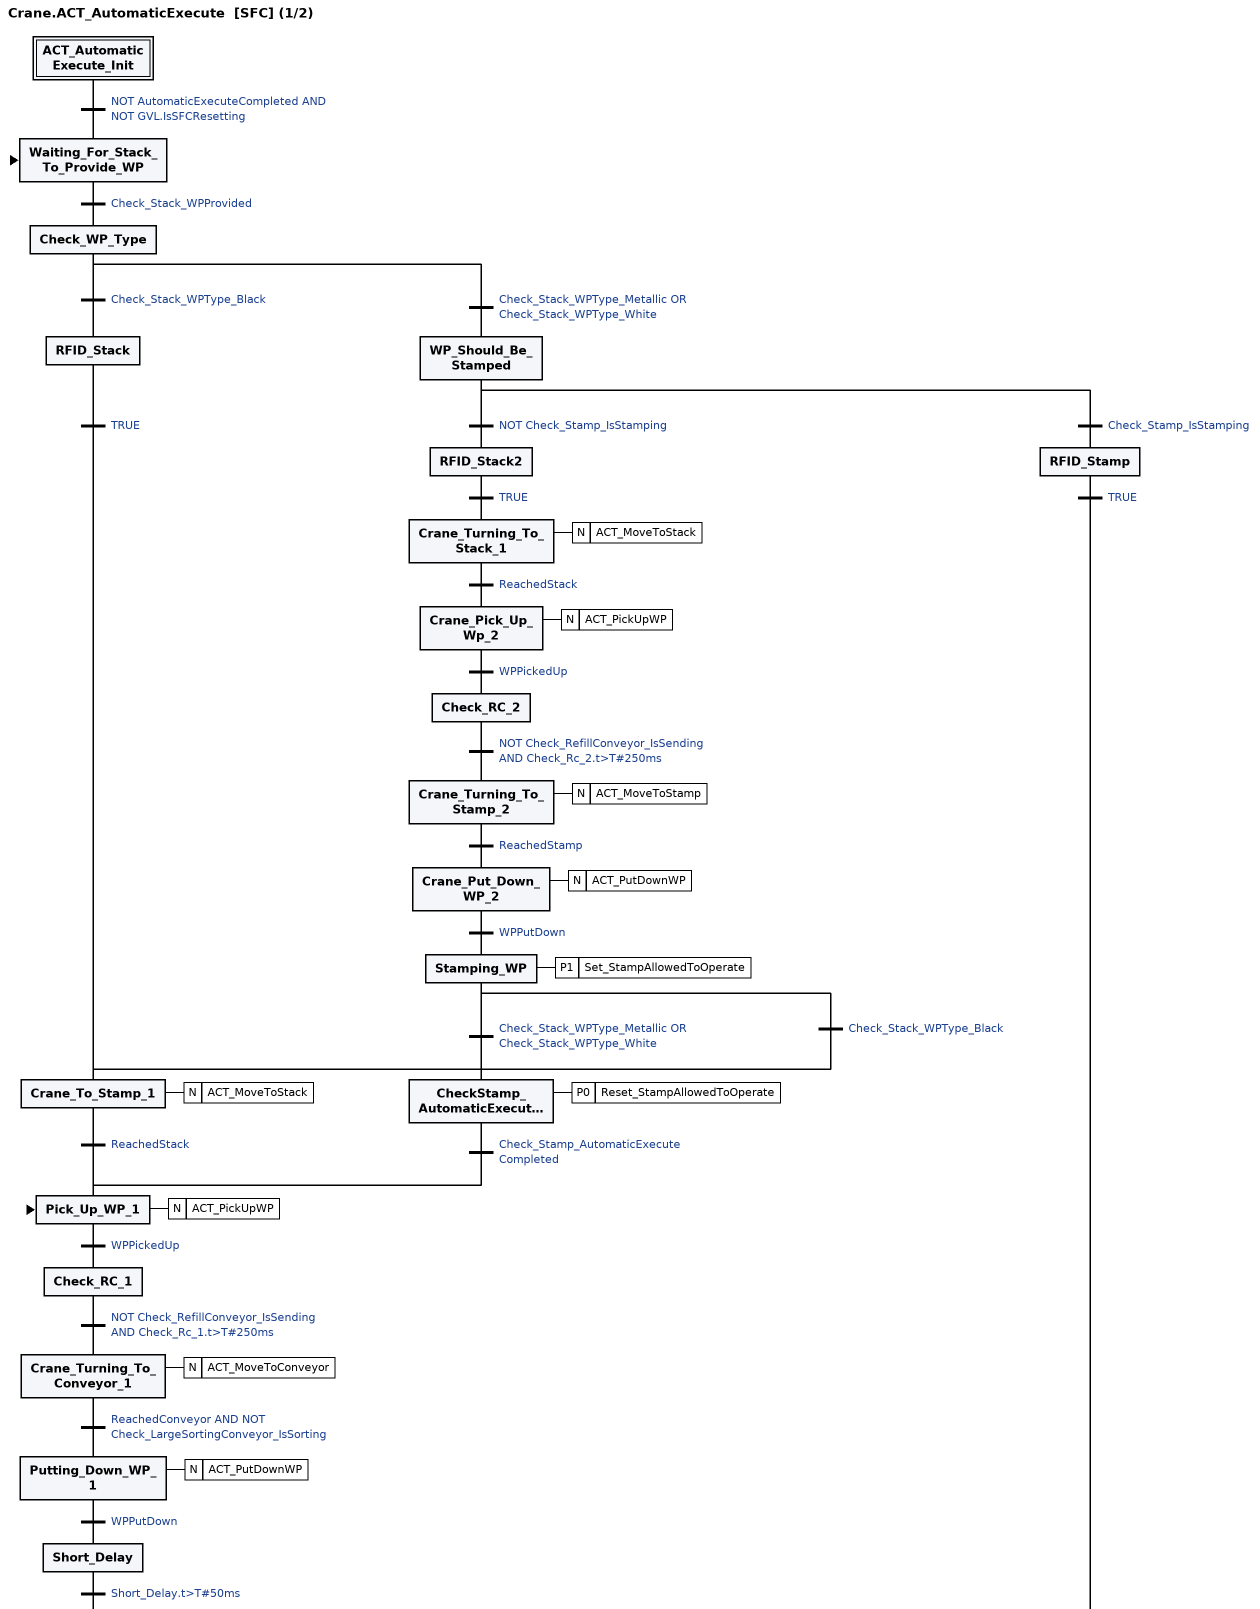
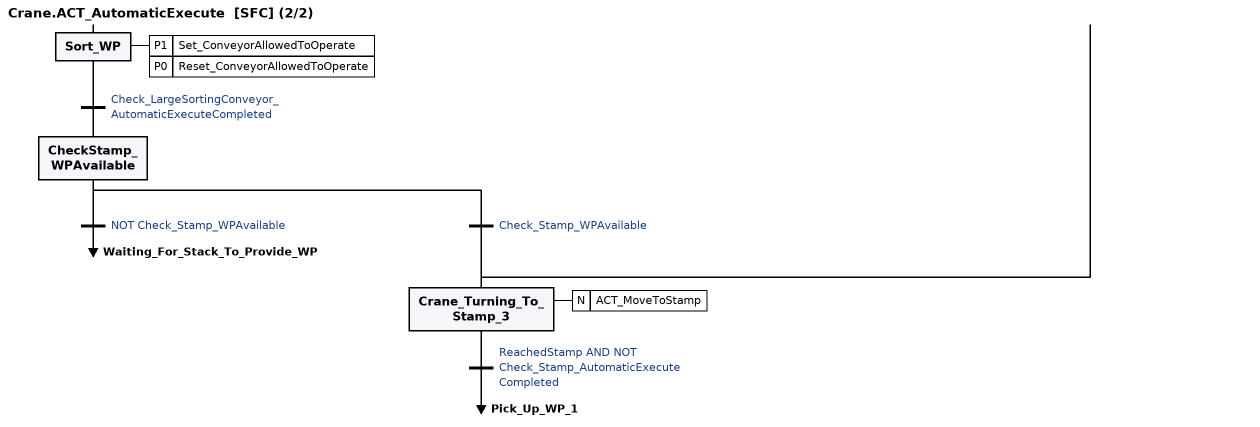
INITIAL_STEP ACT_AutomaticExecute_Init:
END_STEP
TRANSITION FROM ACT_AutomaticExecute_Init TO Waiting_For_Stack_To_Provide_WP
  := NOT AutomaticExecuteCompleted AND NOT GVL.IsSFCResetting;
END_TRANSITION
STEP Waiting_For_Stack_To_Provide_WP:
END_STEP
TRANSITION FROM Waiting_For_Stack_To_Provide_WP TO Check_WP_Type
  := Check_Stack_WPProvided;
END_TRANSITION
STEP Check_WP_Type:
END_STEP
TRANSITION FROM Check_WP_Type TO RFID_Stack
  := Check_Stack_WPType_Black;
END_TRANSITION
TRANSITION FROM Check_WP_Type TO WP_Should_Be_Stamped
  := Check_Stack_WPType_Metallic OR Check_Stack_WPType_White;
END_TRANSITION
STEP RFID_Stack:
END_STEP
TRANSITION FROM RFID_Stack TO Crane_To_Stamp_1
  := TRUE;
END_TRANSITION
STEP Crane_To_Stamp_1:
  ACT_MoveToStack(N);
END_STEP
TRANSITION FROM Crane_To_Stamp_1 TO Pick_Up_WP_1
  := ReachedStack;
END_TRANSITION
STEP Pick_Up_WP_1:
  ACT_PickUpWP(N);
END_STEP
TRANSITION FROM Pick_Up_WP_1 TO Check_RC_1
  := WPPickedUp;
END_TRANSITION
STEP Check_RC_1:
END_STEP
TRANSITION FROM Check_RC_1 TO Crane_Turning_To_Conveyor_1
  := NOT Check_RefillConveyor_IsSending AND Check_Rc_1.t>T#250ms;
END_TRANSITION
STEP Crane_Turning_To_Conveyor_1:
  ACT_MoveToConveyor(N);
END_STEP
TRANSITION FROM Crane_Turning_To_Conveyor_1 TO Putting_Down_WP_1
  := ReachedConveyor AND NOT Check_LargeSortingConveyor_IsSorting;
END_TRANSITION
STEP Putting_Down_WP_1:
  ACT_PutDownWP(N);
END_STEP
TRANSITION FROM Putting_Down_WP_1 TO Short_Delay
  := WPPutDown;
END_TRANSITION
STEP Short_Delay:
END_STEP
TRANSITION FROM Short_Delay TO Sort_WP
  := Short_Delay.t>T#50ms;
END_TRANSITION
STEP Sort_WP:
  Set_ConveyorAllowedToOperate(P1);
  Reset_ConveyorAllowedToOperate(P0);
END_STEP
TRANSITION FROM Sort_WP TO CheckStamp_WPAvailable
  := Check_LargeSortingConveyor_AutomaticExecuteCompleted;
END_TRANSITION
STEP CheckStamp_WPAvailable:
END_STEP
TRANSITION FROM CheckStamp_WPAvailable TO Waiting_For_Stack_To_Provide_WP
  := NOT Check_Stamp_WPAvailable;
END_TRANSITION
TRANSITION FROM CheckStamp_WPAvailable TO Crane_Turning_To_Stamp_3
  := Check_Stamp_WPAvailable;
END_TRANSITION
STEP WP_Should_Be_Stamped:
END_STEP
TRANSITION FROM WP_Should_Be_Stamped TO RFID_Stack2
  := NOT Check_Stamp_IsStamping;
END_TRANSITION
TRANSITION FROM WP_Should_Be_Stamped TO RFID_Stamp
  := Check_Stamp_IsStamping;
END_TRANSITION
STEP RFID_Stack2:
END_STEP
TRANSITION FROM RFID_Stack2 TO Crane_Turning_To_Stack_1
  := TRUE;
END_TRANSITION
STEP Crane_Turning_To_Stack_1:
  ACT_MoveToStack(N);
END_STEP
TRANSITION FROM Crane_Turning_To_Stack_1 TO Crane_Pick_Up_Wp_2
  := ReachedStack;
END_TRANSITION
STEP Crane_Pick_Up_Wp_2:
  ACT_PickUpWP(N);
END_STEP
TRANSITION FROM Crane_Pick_Up_Wp_2 TO Check_RC_2
  := WPPickedUp;
END_TRANSITION
STEP Check_RC_2:
END_STEP
TRANSITION FROM Check_RC_2 TO Crane_Turning_To_Stamp_2
  := NOT Check_RefillConveyor_IsSending AND Check_Rc_2.t>T#250ms;
END_TRANSITION
STEP Crane_Turning_To_Stamp_2:
  ACT_MoveToStamp(N);
END_STEP
TRANSITION FROM Crane_Turning_To_Stamp_2 TO Crane_Put_Down_WP_2
  := ReachedStamp;
END_TRANSITION
STEP Crane_Put_Down_WP_2:
  ACT_PutDownWP(N);
END_STEP
TRANSITION FROM Crane_Put_Down_WP_2 TO Stamping_WP
  := WPPutDown;
END_TRANSITION
STEP Stamping_WP:
  Set_StampAllowedToOperate(P1);
END_STEP
TRANSITION FROM Stamping_WP TO CheckStamp_AutomaticExecuteCompleted
  := Check_Stack_WPType_Metallic OR Check_Stack_WPType_White;
END_TRANSITION
TRANSITION FROM Stamping_WP TO Crane_To_Stamp_1
  := Check_Stack_WPType_Black;
END_TRANSITION
STEP CheckStamp_AutomaticExecuteCompleted:
  Reset_StampAllowedToOperate(P0);
END_STEP
TRANSITION FROM CheckStamp_AutomaticExecuteCompleted TO Pick_Up_WP_1
  := Check_Stamp_AutomaticExecuteCompleted;
END_TRANSITION
STEP RFID_Stamp:
END_STEP
TRANSITION FROM RFID_Stamp TO Crane_Turning_To_Stamp_3
  := TRUE;
END_TRANSITION
STEP Crane_Turning_To_Stamp_3:
  ACT_MoveToStamp(N);
END_STEP
TRANSITION FROM Crane_Turning_To_Stamp_3 TO Pick_Up_WP_1
  := ReachedStamp AND NOT Check_Stamp_AutomaticExecuteCompleted;
END_TRANSITION
END_ACTION

ACTION ACT_EmergencyStop:
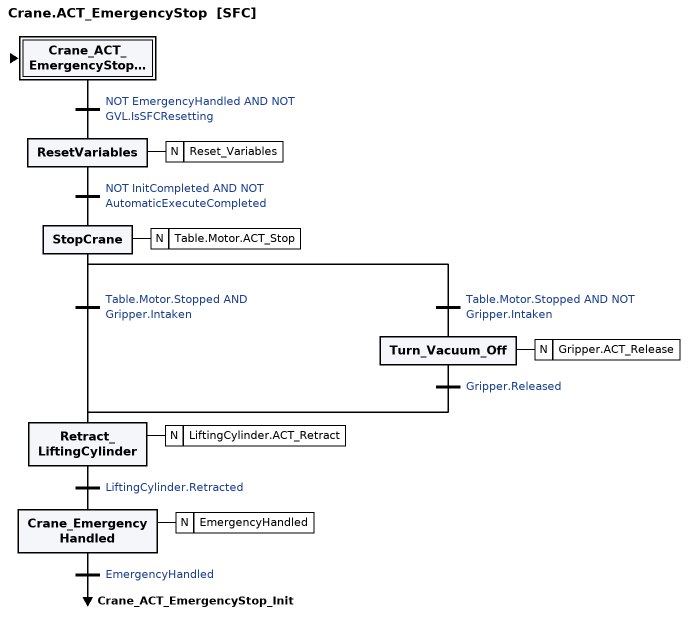
INITIAL_STEP Crane_ACT_EmergencyStop_Init:
END_STEP
TRANSITION FROM Crane_ACT_EmergencyStop_Init TO ResetVariables
  := NOT EmergencyHandled AND NOT GVL.IsSFCResetting;
END_TRANSITION
STEP ResetVariables:
  Reset_Variables(N);
END_STEP
TRANSITION FROM ResetVariables TO StopCrane
  := NOT InitCompleted AND NOT AutomaticExecuteCompleted;
END_TRANSITION
STEP StopCrane:
  Table.Motor.ACT_Stop(N);
END_STEP
TRANSITION FROM StopCrane TO Retract_LiftingCylinder
  := Table.Motor.Stopped AND Gripper.Intaken;
END_TRANSITION
TRANSITION FROM StopCrane TO Turn_Vacuum_Off
  := Table.Motor.Stopped AND NOT Gripper.Intaken;
END_TRANSITION
STEP Turn_Vacuum_Off:
  Gripper.ACT_Release(N);
END_STEP
TRANSITION FROM Turn_Vacuum_Off TO Retract_LiftingCylinder
  := Gripper.Released;
END_TRANSITION
STEP Retract_LiftingCylinder:
  LiftingCylinder.ACT_Retract(N);
END_STEP
TRANSITION FROM Retract_LiftingCylinder TO Crane_EmergencyHandled
  := LiftingCylinder.Retracted;
END_TRANSITION
STEP Crane_EmergencyHandled:
  EmergencyHandled(N);
END_STEP
TRANSITION FROM Crane_EmergencyHandled TO Crane_ACT_EmergencyStop_Init
  := EmergencyHandled;
END_TRANSITION
END_ACTION

ACTION ACT_Init:
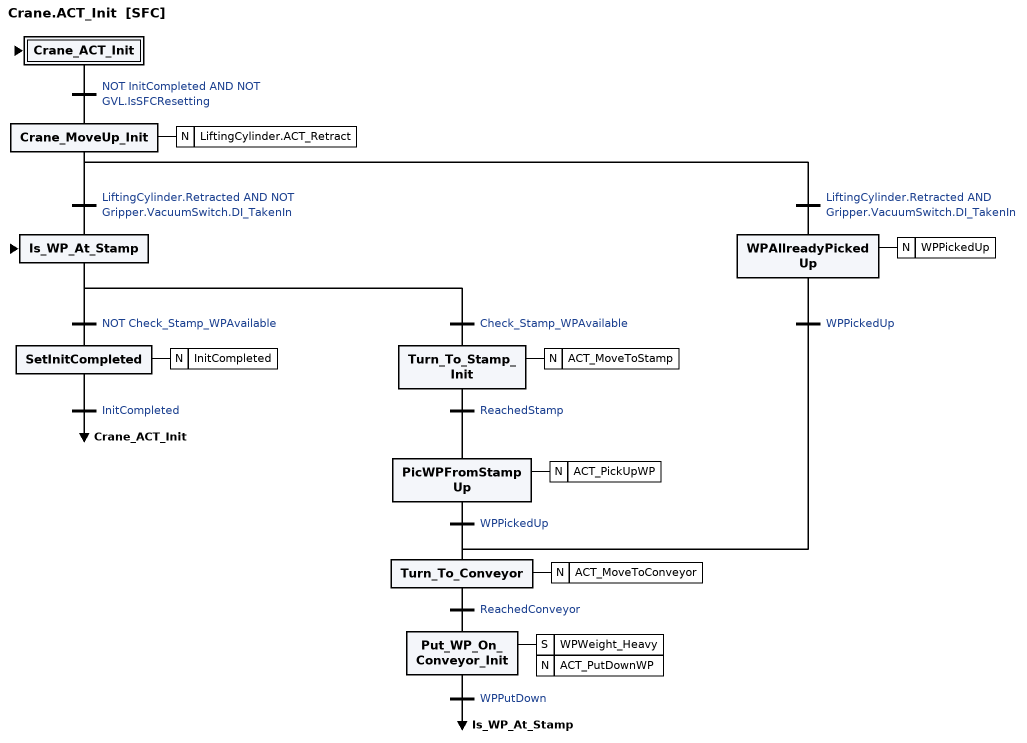
INITIAL_STEP Crane_ACT_Init:
END_STEP
TRANSITION FROM Crane_ACT_Init TO Crane_MoveUp_Init
  := NOT InitCompleted AND NOT GVL.IsSFCResetting;
END_TRANSITION
STEP Crane_MoveUp_Init:
  LiftingCylinder.ACT_Retract(N);
END_STEP
TRANSITION FROM Crane_MoveUp_Init TO Is_WP_At_Stamp
  := LiftingCylinder.Retracted AND NOT Gripper.VacuumSwitch.DI_TakenIn;
END_TRANSITION
TRANSITION FROM Crane_MoveUp_Init TO WPAllreadyPickedUp
  := LiftingCylinder.Retracted AND Gripper.VacuumSwitch.DI_TakenIn;
END_TRANSITION
STEP WPAllreadyPickedUp:
  WPPickedUp(N);
END_STEP
TRANSITION FROM WPAllreadyPickedUp TO Turn_To_Conveyor
  := WPPickedUp;
END_TRANSITION
STEP Turn_To_Conveyor:
  ACT_MoveToConveyor(N);
END_STEP
TRANSITION FROM Turn_To_Conveyor TO Put_WP_On_Conveyor_Init
  := ReachedConveyor;
END_TRANSITION
STEP Put_WP_On_Conveyor_Init:
  WPWeight_Heavy(S);
  ACT_PutDownWP(N);
END_STEP
TRANSITION FROM Put_WP_On_Conveyor_Init TO Is_WP_At_Stamp
  := WPPutDown;
END_TRANSITION
STEP Is_WP_At_Stamp:
END_STEP
TRANSITION FROM Is_WP_At_Stamp TO SetInitCompleted
  := NOT Check_Stamp_WPAvailable;
END_TRANSITION
TRANSITION FROM Is_WP_At_Stamp TO Turn_To_Stamp_Init
  := Check_Stamp_WPAvailable;
END_TRANSITION
STEP Turn_To_Stamp_Init:
  ACT_MoveToStamp(N);
END_STEP
TRANSITION FROM Turn_To_Stamp_Init TO PicWPFromStampUp
  := ReachedStamp;
END_TRANSITION
STEP PicWPFromStampUp:
  ACT_PickUpWP(N);
END_STEP
TRANSITION FROM PicWPFromStampUp TO Turn_To_Conveyor
  := WPPickedUp;
END_TRANSITION
STEP SetInitCompleted:
  InitCompleted(N);
END_STEP
TRANSITION FROM SetInitCompleted TO Crane_ACT_Init
  := InitCompleted;
END_TRANSITION
END_ACTION
END_FUNCTION_BLOCK

FUNCTION_BLOCK EnergyMonitor
VAR_INPUT	
END_VAR
VAR_OUTPUT
END_VAR
VAR
	//Hardware Input Variables
	BK_1_6_Wattmeter : Wattmeter;
	BK_2_3_7_Wattmeter : Wattmeter;
	BK_4_5_8_9_10_11_Wattmeter : Wattmeter;
	
	GearPoint_80l_min : GearPointFlowSensor;
	GearPoint_120l_min : GearPointFlowSensor;
	PressureSensor_4bar : PressureSensor_4bar;
	
	Flow_2to200l_min : FlowSensor;
	Transducer_0to10AC_0to10V : A_to_V_Transducer;
	ExtSensor_0to10V : V_Sensor;
	
	PressureSensor : PressureSensor;
	
	//Hardware Output Variables
	SmallContacter_left : ProtectiveContact;
	SmallContacter_right : ProtectiveContact;
	
	ChangeoverMagnetVaveRelay : MagnetValve;
END_VAR

                  
                
END_FUNCTION_BLOCK

FUNCTION_BLOCK LargeSortingConveyor
VAR_INPUT
	//Hardware
	Panel : OperationPanel;	
	Motor : Motor;
	Seperator1 : MonostableCylinder;
	Seperator2 : MonostableCylinder;	
	PsBeginning : PresenceSensor;		
	OptRamp1 : OpticalSensor;
	IndRamp1 : InductiveSensor;
	Ramp1 : Ramp;
	UltrasonicSensor : UltrasonicSensor;
	Switch : Switch;
	OptRamp2 : OpticalSensor;
	IndRamp2 : InductiveSensor;
	Ramp2 : Ramp;
	OptEnd : OpticalSensor;	
	Ramp3 : Ramp;
	RFID : RFID;
	//NOT USED BUT USABLE
	OptBeginning : OpticalSensor;
	
	//Software
	Check_AllowedToOperate : BOOL;
	Check_FollowConveyorInitCompleted : BOOL;	
	Check_FollowConveyorAutoamticExecuteCompleted : BOOL;	
	Check_EngineStop : BOOL;	
	SFCReset : BOOL;	//Only for SFC implementation
END_VAR
VAR_OUTPUT			
	//Software
	StartButton : BOOL;
	ManuelMode : BOOL;
	AutomaticMode : BOOL;
	InitCompleted : BOOL;
	FollowConveyor_AllowedToInit : BOOL;		
	FollowConveyor_AllowedToOperate : BOOL;	
	NumberOfWPsAtConveyor : USINT;
	AutomaticExecuteCompleted : BOOL;
	EmergencyStop : BOOL;
	EmergencyHandled : BOOL;	
	IsSorting : BOOL;	
END_VAR
VAR	
	//Hardware		
	ConveyorSpeed AT %Q* : INT;
	
	//Software
	WPSorted : BOOL;
	WPTypeChecked : BOOL;
	TargetChanged : BOOL;
	WPType_White : BOOL;
	WPType_Black : BOOL;
	WPType_Metallic : BOOL;
	CurrentTarget_Ramp1 : BOOL;	
	CurrentTarget_Conveyor : BOOL;	
	CurrentTarget_Ramp2 : BOOL;
	CurrentTarget_Ramp3 : BOOL;	
	Priority_White : UINT;
	Priority_Black: UINT;
	Priority_Metallic : UINT;
END_VAR

                  Panel();
ACT_CountWPsAtConveyor();
StartButton := Panel.StartButton;
ManuelMode := Panel.ManuelMode; 
AutomaticMode := Panel.AutomaticMode;
EmergencyStop := Panel.EmergencyStop;
Check_AllowedToOperate := Main.Check_LargeSortingConveyor_AllowedToOperate;
Check_FollowConveyorInitCompleted := Main.Check_LargeSortingConveyor_FollowConveyorInitCompleted;
Check_FollowConveyorAutoamticExecuteCompleted := Main.Check_LargeSortingConveyor_FollowConveyorAutoamticExecuteCompleted;
Check_EngineStop := MAIN.PPU_EngineStop;
IF Check_EngineStop THEN
	Motor.ACT_Stop();
END_IF
                

ACTION Reset_FollowConveyorAllowedToOperate:
                      FollowConveyor_AllowedToOperate := FALSE;
                    
END_ACTION

ACTION Reset_Variables:
                      InitCompleted := FALSE;
FollowConveyor_AllowedToInit := FALSE;
FollowConveyor_AllowedToOperate := FALSE;
AutomaticExecuteCompleted := FALSE;
IsSorting:=FALSE;

WPSorted:=FALSE;
WPTypeChecked:=FALSE;
TargetChanged:=FALSE;
WPType_White:=FALSE;
WPType_Black:=FALSE;
WPType_Metallic:=FALSE;
CurrentTarget_Ramp1:=FALSE;
CurrentTarget_Conveyor:=FALSE;
CurrentTarget_Ramp2:=FALSE;
CurrentTarget_Ramp3:=FALSE;
                    
END_ACTION

ACTION Set_FollowConveyorAllowedToOperate:
                      FollowConveyor_AllowedToOperate := TRUE;
                    
END_ACTION

ACTION Set_OneWP:
                      NumberOfWPsAtConveyor:=1;
                    
END_ACTION

ACTION Set_PriorityBlack:
                      Priority_Black := 4;
                    
END_ACTION

ACTION Set_PriorityMetallic:
                      Priority_Metallic := 3;
                    
END_ACTION

ACTION Set_PriorityWhite:
                      Priority_White := 1;
                    
END_ACTION

ACTION Set_ThreeWP:
                      NumberOfWPsAtConveyor:=3;
                    
END_ACTION

ACTION Set_TwoWP:
                      NumberOfWPsAtConveyor:=2;
                    
END_ACTION

ACTION Set_ZeroWP:
                      NumberOfWPsAtConveyor:=0;
                    
END_ACTION

ACTION ACT_ChangeTarget:
